LIN {X 0,Y 448.78,Z 726.193,A -85,B 0,C 180,E1 -8884.616,E2 -8884.616} C_VEL
LIN {X 0,Y 448.11,Z 736.801,A -85,B 0,C 180,E1 -8885.667,E2 -8885.667} C_VEL
LIN {X 0,Y 447.551,Z 746.669,A -85,B 0,C 180,E1 -8886.885,E2 -8886.885} C_VEL
LIN {X 0,Y 447.034,Z 755.083,A -85,B 0,C 180,E1 -8888.183,E2 -8888.183} C_VEL
LIN {X 0,Y 446.974,Z 755.977,A -85,B 0,C 180,E1 -8888.339,E2 -8888.339} C_VEL
LIN {X 0,Y 446.099,Z 759.432,A -85,B 0,C 180,E1 -8888.947,E2 -8888.947} C_VEL
LIN {X 0,Y 442.936,Z 764.696,A -85,B 0,C 180,E1 -8889.952,E2 -8889.952} C_VEL
LIN {X 0,Y 439.821,Z 769.35,A -85,B 0,C 180,E1 -8891.018,E2 -8891.018} C_VEL
LIN {X 0,Y 439.028,Z 771.716,A -85,B 0,C 180,E1 -8891.713,E2 -8891.713} C_VEL
LIN {X 0,Y 438.819,Z 775.806,A -85,B 0,C 180,E1 -8893.245,E2 -8893.245} C_VEL
LIN {X 0,Y 438.678,Z 777.727,A -85,B 0,C 180,E1 -8894.196,E2 -8894.196} C_VEL
LIN {X 0,Y 438.549,Z 779.208,A -85,B 0,C 180,E1 -8895.143,E2 -8895.143} C_VEL
LIN {X 0,Y 438.47,Z 780.829,A -85,B 0,C 180,E1 -8897.033,E2 -8897.033} C_VEL
LIN {X 0,Y 438.51,Z 781.044,A -85,B 0,C 180,E1 -8897.975,E2 -8897.975} C_VEL
LIN {X 0,Y 438.515,Z 780.818,A -85,B 0,C 180,E1 -8898.912,E2 -8898.912} C_VEL
LIN {X 0,Y 438.516,Z 779.204,A -85,B 0,C 180,E1 -8900.778,E2 -8900.778} C_VEL
LIN {X 0,Y 438.62,Z 777.768,A -85,B 0,C 180,E1 -8901.709,E2 -8901.709} C_VEL
LIN {X 0,Y 438.838,Z 774.591,A -85,B 0,C 180,E1 -8903.185,E2 -8903.185} C_VEL
LIN {X 0,Y 439.068,Z 769.268,A -85,B 0,C 180,E1 -8904.949,E2 -8904.949} C_VEL
LIN {X 0,Y 439.407,Z 762.676,A -85,B 0,C 180,E1 -8906.562,E2 -8906.562} C_VEL
LIN {X 0,Y 439.846,Z 755.516,A -85,B 0,C 180,E1 -8907.94,E2 -8907.94} C_VEL
LIN {X 0,Y 440.286,Z 748.225,A -85,B 0,C 180,E1 -8909.085,E2 -8909.085} C_VEL
LIN {X 0,Y 440.868,Z 739.403,A -85,B 0,C 180,E1 -8910.228,E2 -8910.228} C_VEL
LIN {X 0,Y 441.415,Z 728.463,A -85,B 0,C 180,E1 -8911.368,E2 -8911.368} C_VEL
LIN {X 0,Y 442.038,Z 717.473,A -85,B 0,C 180,E1 -8912.278,E2 -8912.278} C_VEL
LIN {X 0,Y 442.582,Z 705,A -85,B 0,C 180,E1 -8913.072,E2 -8913.072} C_VEL
LIN {X 0,Y 442.948,Z 692.395,A -85,B 0,C 180,E1 -8913.667,E2 -8913.667} C_VEL
LIN {X 0,Y 443.227,Z 680.1,A -85,B 0,C 180,E1 -8914.063,E2 -8914.063} C_VEL
LIN {X 0,Y 443.477,Z 656.155,A -85,B 0,C 180,E1 -8914.488,E2 -8914.488} C_VEL
LIN {X 0,Y 444.044,Z 588.908,A -85,B 0,C 180,E1 -8915.579,E2 -8915.579} C_VEL
LIN {X 0,Y 439.593,Z 575.73,A -85,B 0,C 180,E1 -8915.994,E2 -8915.994} C_VEL
LIN {X 0,Y 439.534,Z 575.738,A -85,B 0,C 180,E1 -8918.274,E2 -8918.274} C_VEL
LIN {X 0,Y 439.51,Z 575.741,A -85,B 0,C 180,E1 -8921.998,E2 -8921.998} C_VEL
LIN {X 0,Y 439.464,Z 575.743,A -85,B 0,C 180,E1 -8925.775,E2 -8925.775} C_VEL
LIN {X 0,Y 439.443,Z 575.743,A -85,B 0,C 180,E1 -8929.337,E2 -8929.337} C_VEL
LIN {X 0,Y 439.365,Z 575.754,A -85,B 0,C 180,E1 -8932.575,E2 -8932.575} C_VEL
LIN {X 0,Y 439.397,Z 575.751,A -85,B 0,C 180,E1 -8935.585,E2 -8935.585} C_VEL
LIN {X 0,Y 439.469,Z 575.744,A -85,B 0,C 180,E1 -8938.02,E2 -8938.02} C_VEL
LIN {X 0,Y 444.266,Z 589.404,A -85,B 0,C 180,E1 -8938.464,E2 -8938.464} C_VEL
LIN {X 0,Y 443.152,Z 678.564,A -85,B 0,C 180,E1 -8939.987,E2 -8939.987} C_VEL
LIN {X 0,Y 442.929,Z 692.439,A -85,B 0,C 180,E1 -8940.431,E2 -8940.431} C_VEL
LIN {X 0,Y 442.524,Z 705.387,A -85,B 0,C 180,E1 -8941.049,E2 -8941.049} C_VEL
LIN {X 0,Y 442.045,Z 716.757,A -85,B 0,C 180,E1 -8941.778,E2 -8941.778} C_VEL
LIN {X 0,Y 441.489,Z 728.769,A -85,B 0,C 180,E1 -8942.767,E2 -8942.767} C_VEL
LIN {X 0,Y 440.928,Z 738.453,A -85,B 0,C 180,E1 -8943.77,E2 -8943.77} C_VEL
LIN {X 0,Y 440.317,Z 748.569,A -85,B 0,C 180,E1 -8945.071,E2 -8945.071} C_VEL
LIN {X 0,Y 439.875,Z 755.956,A -85,B 0,C 180,E1 -8946.238,E2 -8946.238} C_VEL
LIN {X 0,Y 439.396,Z 763.311,A -85,B 0,C 180,E1 -8947.662,E2 -8947.662} C_VEL
LIN {X 0,Y 439.083,Z 769.474,A -85,B 0,C 180,E1 -8949.192,E2 -8949.192} C_VEL
LIN {X 0,Y 438.838,Z 773.436,A -85,B 0,C 180,E1 -8950.436,E2 -8950.436} C_VEL
LIN {X 0,Y 438.69,Z 776.55,A -85,B 0,C 180,E1 -8951.69,E2 -8951.69} C_VEL
LIN {X 0,Y 438.577,Z 778.129,A -85,B 0,C 180,E1 -8952.512,E2 -8952.512} C_VEL
LIN {X 0,Y 438.477,Z 779.994,A -85,B 0,C 180,E1 -8953.84,E2 -8953.84} C_VEL
LIN {X 0,Y 438.416,Z 780.98,A -85,B 0,C 180,E1 -8955.143,E2 -8955.143} C_VEL
LIN {X 0,Y 438.403,Z 781.18,A -85,B 0,C 180,E1 -8956.423,E2 -8956.423} C_VEL
LIN {X 0,Y 438.468,Z 780.644,A -85,B 0,C 180,E1 -8957.685,E2 -8957.685} C_VEL
LIN {X 0,Y 438.56,Z 779.387,A -85,B 0,C 180,E1 -8958.926,E2 -8958.926} C_VEL
LIN {X 0,Y 438.764,Z 775.998,A -85,B 0,C 180,E1 -8960.807,E2 -8960.807} C_VEL
LIN {X 0,Y 439.01,Z 772.573,A -85,B 0,C 180,E1 -8962.11,E2 -8962.11} C_VEL
LIN {X 0,Y 439.311,Z 767.045,A -85,B 0,C 180,E1 -8963.707,E2 -8963.707} C_VEL
LIN {X 0,Y 439.69,Z 760.584,A -85,B 0,C 180,E1 -8965.15,E2 -8965.15} C_VEL
LIN {X 0,Y 440.113,Z 753.59,A -85,B 0,C 180,E1 -8966.403,E2 -8966.403} C_VEL
LIN {X 0,Y 440.746,Z 744.764,A -85,B 0,C 180,E1 -8967.683,E2 -8967.683} C_VEL
LIN {X 0,Y 441.288,Z 735.189,A -85,B 0,C 180,E1 -8968.814,E2 -8968.814} C_VEL
LIN {X 0,Y 441.891,Z 724.799,A -85,B 0,C 180,E1 -8969.803,E2 -8969.803} C_VEL
LIN {X 0,Y 442.376,Z 714.046,A -85,B 0,C 180,E1 -8970.619,E2 -8970.619} C_VEL
LIN {X 0,Y 442.917,Z 701.443,A -85,B 0,C 180,E1 -8971.355,E2 -8971.355} C_VEL
LIN {X 0,Y 443.186,Z 688.797,A -85,B 0,C 180,E1 -8971.893,E2 -8971.893} C_VEL
LIN {X 0,Y 443.426,Z 676.012,A -85,B 0,C 180,E1 -8972.239,E2 -8972.239} C_VEL
LIN {X 0,Y 444.343,Z 588.817,A -85,B 0,C 180,E1 -8973.74,E2 -8973.74} C_VEL
LIN {X 0,Y 439.477,Z 575.744,A -85,B 0,C 180,E1 -8974.203,E2 -8974.203} C_VEL
LIN {X 0,Y 439.357,Z 575.757,A -85,B 0,C 180,E1 -8977.424,E2 -8977.424} C_VEL
LIN {X 0,Y 439.433,Z 575.75,A -85,B 0,C 180,E1 -8980.662,E2 -8980.662} C_VEL
LIN {X 0,Y 439.453,Z 575.747,A -85,B 0,C 180,E1 -8984.224,E2 -8984.224} C_VEL
LIN {X 0,Y 439.503,Z 575.739,A -85,B 0,C 180,E1 -8988.002,E2 -8988.002} C_VEL
LIN {X 0,Y 439.539,Z 575.732,A -85,B 0,C 180,E1 -8991.726,E2 -8991.726} C_VEL
LIN {X 0,Y 439.618,Z 575.726,A -85,B 0,C 180,E1 -8994.496,E2 -8994.496} C_VEL
LIN {X 0,Y 439.626,Z 575.721,A -85,B 0,C 180,E1 -8998.168,E2 -8998.168} C_VEL
LIN {X 0,Y 439.755,Z 575.706,A -85,B 0,C 180,E1 -9000,E2 -9000} C_VEL
LIN {X 0,Y 439.648,Z 575.719,A -85,B 0,C 180,E1 -9002.749,E2 -9002.749} C_VEL
LIN {X 0,Y 439.613,Z 575.724,A -85,B 0,C 180,E1 -9006.425,E2 -9006.425} C_VEL
LIN {X 0,Y 439.492,Z 575.734,A -85,B 0,C 180,E1 -9009.202,E2 -9009.202} C_VEL
LIN {X 0,Y 439.495,Z 575.734,A -85,B 0,C 180,E1 -9012.727,E2 -9012.727} C_VEL
LIN {X 0,Y 439.438,Z 575.744,A -85,B 0,C 180,E1 -9016.349,E2 -9016.349} C_VEL
LIN {X 0,Y 439.395,Z 575.745,A -85,B 0,C 180,E1 -9019.627,E2 -9019.627} C_VEL
LIN {X 0,Y 439.359,Z 575.757,A -85,B 0,C 180,E1 -9022.576,E2 -9022.576} C_VEL
LIN {X 0,Y 439.398,Z 575.748,A -85,B 0,C 180,E1 -9025.585,E2 -9025.585} C_VEL
LIN {X 0,Y 439.418,Z 575.752,A -85,B 0,C 180,E1 -9028.674,E2 -9028.674} C_VEL
LIN {X 0,Y 439.368,Z 575.753,A -85,B 0,C 180,E1 -9031.861,E2 -9031.861} C_VEL
LIN {X 0,Y 439.395,Z 575.75,A -85,B 0,C 180,E1 -9035.157,E2 -9035.157} C_VEL
LIN {X 0,Y 439.394,Z 575.753,A -85,B 0,C 180,E1 -9038.594,E2 -9038.594} C_VEL
LIN {X 0,Y 439.4,Z 575.747,A -85,B 0,C 180,E1 -9041.26,E2 -9041.26} C_VEL
LIN {X 0,Y 439.404,Z 575.754,A -85,B 0,C 180,E1 -9044.729,E2 -9044.729} C_VEL
LIN {X 0,Y 439.393,Z 575.751,A -85,B 0,C 180,E1 -9047.797,E2 -9047.797} C_VEL
LIN {X 0,Y 439.448,Z 575.747,A -85,B 0,C 180,E1 -9050.231,E2 -9050.231} C_VEL
LIN {X 0,Y 439.374,Z 575.753,A -85,B 0,C 180,E1 -9053.714,E2 -9053.714} C_VEL
LIN {X 0,Y 439.371,Z 575.755,A -85,B 0,C 180,E1 -9057.055,E2 -9057.055} C_VEL
LIN {X 0,Y 439.443,Z 575.82,A -85,B 0,C 180,E1 -9060.707,E2 -9060.707} C_VEL
LIN {X 0,Y 442.42,Z 589.659,A -85,B 0,C 180,E1 -9063.274,E2 -9063.274} C_VEL
LIN {X 0,Y 442.893,Z 594.558,A -85,B 0,C 180,E1 -9064.128,E2 -9064.128} C_VEL
LIN {X 0,Y 441.873,Z 612.173,A -85,B 0,C 180,E1 -9067.021,E2 -9067.021} C_VEL
LIN {X 0,Y 440.837,Z 633.371,A -85,B 0,C 180,E1 -9070.441,E2 -9070.441} C_VEL
LIN {X 0,Y 440.413,Z 641.915,A -85,B 0,C 180,E1 -9071.806,E2 -9071.806} C_VEL
LIN {X 0,Y 443.891,Z 669.193,A -85,B 0,C 180,E1 -9072.436,E2 -9072.436} C_VEL
LIN {X 0,Y 442.998,Z 751.905,A -85,B 0,C 180,E1 -9073.852,E2 -9073.852} C_VEL
LIN {X 0,Y 442.553,Z 765.081,A -85,B 0,C 180,E1 -9074.249,E2 -9074.249} C_VEL
LIN {X 0,Y 442.027,Z 776.143,A -85,B 0,C 180,E1 -9074.732,E2 -9074.732} C_VEL
LIN {X 0,Y 441.373,Z 788.842,A -85,B 0,C 180,E1 -9075.476,E2 -9075.476} C_VEL
LIN {X 0,Y 440.764,Z 800.147,A -85,B 0,C 180,E1 -9076.344,E2 -9076.344} C_VEL
LIN {X 0,Y 440.178,Z 811.45,A -85,B 0,C 180,E1 -9077.436,E2 -9077.436} C_VEL
LIN {X 0,Y 439.622,Z 820.217,A -85,B 0,C 180,E1 -9078.473,E2 -9078.473} C_VEL
LIN {X 0,Y 439.176,Z 828.317,A -85,B 0,C 180,E1 -9079.629,E2 -9079.629} C_VEL
LIN {X 0,Y 438.816,Z 836.256,A -85,B 0,C 180,E1 -9081.016,E2 -9081.016} C_VEL
LIN {X 0,Y 438.608,Z 843.573,A -85,B 0,C 180,E1 -9082.635,E2 -9082.635} C_VEL
LIN {X 0,Y 438.479,Z 847.975,A -85,B 0,C 180,E1 -9083.869,E2 -9083.869} C_VEL
LIN {X 0,Y 438.401,Z 852.206,A -85,B 0,C 180,E1 -9085.403,E2 -9085.403} C_VEL
LIN {X 0,Y 438.479,Z 854.154,A -85,B 0,C 180,E1 -9086.324,E2 -9086.324} C_VEL
LIN {X 0,Y 438.509,Z 855.616,A -85,B 0,C 180,E1 -9087.244,E2 -9087.244} C_VEL
LIN {X 0,Y 438.466,Z 856.659,A -85,B 0,C 180,E1 -9088.163,E2 -9088.163} C_VEL
LIN {X 0,Y 438.381,Z 857.299,A -85,B 0,C 180,E1 -9089.081,E2 -9089.081} C_VEL
LIN {X 0,Y 438.361,Z 857.538,A -85,B 0,C 180,E1 -9090,E2 -9090} C_VEL
LIN {X 0,Y 438.466,Z 856.734,A -85,B 0,C 180,E1 -9091.837,E2 -9091.837} C_VEL
LIN {X 0,Y 438.508,Z 855.731,A -85,B 0,C 180,E1 -9092.756,E2 -9092.756} C_VEL
LIN {X 0,Y 438.476,Z 854.299,A -85,B 0,C 180,E1 -9093.676,E2 -9093.676} C_VEL
LIN {X 0,Y 438.453,Z 851.302,A -85,B 0,C 180,E1 -9095.058,E2 -9095.058} C_VEL
LIN {X 0,Y 438.506,Z 847.237,A -85,B 0,C 180,E1 -9096.441,E2 -9096.441} C_VEL
LIN {X 0,Y 438.671,Z 840.963,A -85,B 0,C 180,E1 -9098.058,E2 -9098.058} C_VEL
LIN {X 0,Y 438.909,Z 834.122,A -85,B 0,C 180,E1 -9099.446,E2 -9099.446} C_VEL
LIN {X 0,Y 439.357,Z 825.638,A -85,B 0,C 180,E1 -9100.833,E2 -9100.833} C_VEL
LIN {X 0,Y 439.809,Z 816.892,A -85,B 0,C 180,E1 -9101.989,E2 -9101.989} C_VEL
LIN {X 0,Y 440.399,Z 806.912,A -85,B 0,C 180,E1 -9103.068,E2 -9103.068} C_VEL
LIN {X 0,Y 441.032,Z 795.466,A -85,B 0,C 180,E1 -9104.064,E2 -9104.064} C_VEL
LIN {X 0,Y 441.689,Z 783.61,A -85,B 0,C 180,E1 -9104.867,E2 -9104.867} C_VEL
LIN {X 0,Y 442.214,Z 771.308,A -85,B 0,C 180,E1 -9105.497,E2 -9105.497} C_VEL
LIN {X 0,Y 442.8,Z 757.864,A -85,B 0,C 180,E1 -9105.978,E2 -9105.978} C_VEL
LIN {X 0,Y 443.127,Z 742.721,A -85,B 0,C 180,E1 -9106.291,E2 -9106.291} C_VEL
LIN {X 0,Y 443.758,Z 666.118,A -85,B 0,C 180,E1 -9107.584,E2 -9107.584} C_VEL
LIN {X 0,Y 440.913,Z 642.526,A -85,B 0,C 180,E1 -9108.115,E2 -9108.115} C_VEL
LIN {X 0,Y 441.932,Z 622.104,A -85,B 0,C 180,E1 -9110.966,E2 -9110.966} C_VEL
LIN {X 0,Y 443.256,Z 598.165,A -85,B 0,C 180,E1 -9114.345,E2 -9114.345} C_VEL
LIN {X 0,Y 443.448,Z 594.812,A -85,B 0,C 180,E1 -9114.822,E2 -9114.822} C_VEL
LIN {X 0,Y 441.817,Z 585.976,A -85,B 0,C 180,E1 -9116.194,E2 -9116.194} C_VEL
LIN {X 0,Y 439.473,Z 575.746,A -85,B 0,C 180,E1 -9117.866,E2 -9117.866} C_VEL
LIN {X 0,Y 439.36,Z 575.755,A -85,B 0,C 180,E1 -9120.788,E2 -9120.788} C_VEL
LIN {X 0,Y 439.386,Z 575.756,A -85,B 0,C 180,E1 -9124.043,E2 -9124.043} C_VEL
LIN {X 0,Y 439.361,Z 575.755,A -85,B 0,C 180,E1 -9127.433,E2 -9127.433} C_VEL
LIN {X 0,Y 439.423,Z 575.749,A -85,B 0,C 180,E1 -9129.852,E2 -9129.852} C_VEL
LIN {X 0,Y 439.378,Z 575.752,A -85,B 0,C 180,E1 -9132.626,E2 -9132.626} C_VEL
LIN {X 0,Y 439.399,Z 575.748,A -85,B 0,C 180,E1 -9136.033,E2 -9136.033} C_VEL
LIN {X 0,Y 439.395,Z 575.747,A -85,B 0,C 180,E1 -9139.021,E2 -9139.021} C_VEL
LIN {X 0,Y 439.387,Z 575.747,A -85,B 0,C 180,E1 -9141.604,E2 -9141.604} C_VEL
LIN {X 0,Y 439.394,Z 575.741,A -85,B 0,C 180,E1 -9144.843,E2 -9144.843} C_VEL
LIN {X 0,Y 439.381,Z 575.755,A -85,B 0,C 180,E1 -9148.14,E2 -9148.14} C_VEL
LIN {X 0,Y 439.418,Z 575.736,A -85,B 0,C 180,E1 -9151.326,E2 -9151.326} C_VEL
LIN {X 0,Y 439.398,Z 575.754,A -85,B 0,C 180,E1 -9154.415,E2 -9154.415} C_VEL
LIN {X 0,Y 439.356,Z 575.742,A -85,B 0,C 180,E1 -9157.424,E2 -9157.424} C_VEL
LIN {X 0,Y 439.433,Z 575.748,A -85,B 0,C 180,E1 -9160.662,E2 -9160.662} C_VEL
LIN {X 0,Y 439.453,Z 575.734,A -85,B 0,C 180,E1 -9164.224,E2 -9164.224} C_VEL
LIN {X 0,Y 439.475,Z 575.74,A -85,B 0,C 180,E1 -9168.001,E2 -9168.001} C_VEL
LIN {X 0,Y 439.538,Z 575.72,A -85,B 0,C 180,E1 -9171.726,E2 -9171.726} C_VEL
LIN {X 0,Y 439.619,Z 575.725,A -85,B 0,C 180,E1 -9174.496,E2 -9174.496} C_VEL
LIN {X 0,Y 439.627,Z 575.712,A -85,B 0,C 180,E1 -9178.168,E2 -9178.168} C_VEL
LIN {X 0,Y 439.755,Z 575.698,A -85,B 0,C 180,E1 -9180,E2 -9180} C_VEL
LIN {X 0,Y 439.648,Z 575.722,A -85,B 0,C 180,E1 -9182.749,E2 -9182.749} C_VEL
LIN {X 0,Y 439.611,Z 575.712,A -85,B 0,C 180,E1 -9186.425,E2 -9186.425} C_VEL
LIN {X 0,Y 439.491,Z 575.739,A -85,B 0,C 180,E1 -9189.202,E2 -9189.202} C_VEL
LIN {X 0,Y 439.457,Z 575.736,A -85,B 0,C 180,E1 -9192.938,E2 -9192.938} C_VEL
LIN {X 0,Y 439.438,Z 575.744,A -85,B 0,C 180,E1 -9196.349,E2 -9196.349} C_VEL
LIN {X 0,Y 439.394,Z 575.745,A -85,B 0,C 180,E1 -9199.627,E2 -9199.627} C_VEL
LIN {X 0,Y 439.356,Z 575.756,A -85,B 0,C 180,E1 -9202.576,E2 -9202.576} C_VEL
LIN {X 0,Y 439.398,Z 575.748,A -85,B 0,C 180,E1 -9205.585,E2 -9205.585} C_VEL
LIN {X 0,Y 439.418,Z 575.748,A -85,B 0,C 180,E1 -9208.674,E2 -9208.674} C_VEL
LIN {X 0,Y 439.378,Z 575.751,A -85,B 0,C 180,E1 -9212.034,E2 -9212.034} C_VEL
LIN {X 0,Y 439.39,Z 575.753,A -85,B 0,C 180,E1 -9215.341,E2 -9215.341} C_VEL
LIN {X 0,Y 439.387,Z 575.751,A -85,B 0,C 180,E1 -9218.595,E2 -9218.595} C_VEL
LIN {X 0,Y 439.393,Z 575.738,A -85,B 0,C 180,E1 -9221.259,E2 -9221.259} C_VEL
LIN {X 0,Y 439.401,Z 575.749,A -85,B 0,C 180,E1 -9224.73,E2 -9224.73} C_VEL
LIN {X 0,Y 439.392,Z 575.742,A -85,B 0,C 180,E1 -9227.796,E2 -9227.796} C_VEL
LIN {X 0,Y 439.423,Z 575.746,A -85,B 0,C 180,E1 -9230.228,E2 -9230.228} C_VEL
LIN {X 0,Y 439.375,Z 575.756,A -85,B 0,C 180,E1 -9233.714,E2 -9233.714} C_VEL
LIN {X 0,Y 439.371,Z 575.756,A -85,B 0,C 180,E1 -9237.055,E2 -9237.055} C_VEL
LIN {X 0,Y 439.39,Z 575.754,A -85,B 0,C 180,E1 -9239.824,E2 -9239.824} C_VEL
LIN {X 0,Y 441.332,Z 580.971,A -85,B 0,C 180,E1 -9240.019,E2 -9240.019} C_VEL
LIN {X 0,Y 444.652,Z 589.408,A -85,B 0,C 180,E1 -9240.32,E2 -9240.32} C_VEL
LIN {X 0,Y 443.622,Z 677.951,A -85,B 0,C 180,E1 -9241.785,E2 -9241.785} C_VEL
LIN {X 0,Y 443.413,Z 690.45,A -85,B 0,C 180,E1 -9242.156,E2 -9242.156} C_VEL
LIN {X 0,Y 443.099,Z 702.807,A -85,B 0,C 180,E1 -9242.706,E2 -9242.706} C_VEL
LIN {X 0,Y 442.623,Z 713.699,A -85,B 0,C 180,E1 -9243.357,E2 -9243.357} C_VEL
LIN {X 0,Y 442.044,Z 724.739,A -85,B 0,C 180,E1 -9244.201,E2 -9244.201} C_VEL
LIN {X 0,Y 441.44,Z 734.788,A -85,B 0,C 180,E1 -9245.159,E2 -9245.159} C_VEL
LIN {X 0,Y 440.852,Z 744.173,A -85,B 0,C 180,E1 -9246.264,E2 -9246.264} C_VEL
LIN {X 0,Y 440.29,Z 752.531,A -85,B 0,C 180,E1 -9247.475,E2 -9247.475} C_VEL
LIN {X 0,Y 439.771,Z 760.635,A -85,B 0,C 180,E1 -9248.927,E2 -9248.927} C_VEL
LIN {X 0,Y 439.339,Z 767.04,A -85,B 0,C 180,E1 -9250.371,E2 -9250.371} C_VEL
LIN {X 0,Y 439.028,Z 771.716,A -85,B 0,C 180,E1 -9251.713,E2 -9251.713} C_VEL
LIN {X 0,Y 438.246,Z 773.899,A -85,B 0,C 180,E1 -9252.423,E2 -9252.423} C_VEL
LIN {X 0,Y 435.194,Z 776.991,A -85,B 0,C 180,E1 -9253.594,E2 -9253.594} C_VEL
LIN {X 0,Y 432.653,Z 778.955,A -85,B 0,C 180,E1 -9254.558,E2 -9254.558} C_VEL
LIN {X 0,Y 431.552,Z 780.087,A -85,B 0,C 180,E1 -9255.316,E2 -9255.316} C_VEL
LIN {X 0,Y 431.456,Z 780.354,A -85,B 0,C 180,E1 -9255.575,E2 -9255.575} C_VEL
LIN {X 0,Y 431.395,Z 781.35,A -85,B 0,C 180,E1 -9256.816,E2 -9256.816} C_VEL
LIN {X 0,Y 431.433,Z 781.628,A -85,B 0,C 180,E1 -9257.795,E2 -9257.795} C_VEL
LIN {X 0,Y 431.445,Z 781.506,A -85,B 0,C 180,E1 -9258.728,E2 -9258.728} C_VEL
LIN {X 0,Y 431.437,Z 780.007,A -85,B 0,C 180,E1 -9260.625,E2 -9260.625} C_VEL
LIN {X 0,Y 431.529,Z 778.669,A -85,B 0,C 180,E1 -9261.572,E2 -9261.572} C_VEL
LIN {X 0,Y 431.778,Z 775.393,A -85,B 0,C 180,E1 -9263.165,E2 -9263.165} C_VEL
LIN {X 0,Y 432.001,Z 770.432,A -85,B 0,C 180,E1 -9264.867,E2 -9264.867} C_VEL
LIN {X 0,Y 432.273,Z 765.064,A -85,B 0,C 180,E1 -9266.271,E2 -9266.271} C_VEL
LIN {X 0,Y 432.739,Z 758.341,A -85,B 0,C 180,E1 -9267.673,E2 -9267.673} C_VEL
LIN {X 0,Y 433.251,Z 749.932,A -85,B 0,C 180,E1 -9269.071,E2 -9269.071} C_VEL
LIN {X 0,Y 433.838,Z 741.33,A -85,B 0,C 180,E1 -9270.232,E2 -9270.232} C_VEL
LIN {X 0,Y 434.416,Z 730.777,A -85,B 0,C 180,E1 -9271.391,E2 -9271.391} C_VEL
LIN {X 0,Y 435.012,Z 720.168,A -85,B 0,C 180,E1 -9272.315,E2 -9272.315} C_VEL
LIN {X 0,Y 435.616,Z 708.398,A -85,B 0,C 180,E1 -9273.121,E2 -9273.121} C_VEL
LIN {X 0,Y 436.035,Z 696.124,A -85,B 0,C 180,E1 -9273.754,E2 -9273.754} C_VEL
LIN {X 0,Y 436.328,Z 683.342,A -85,B 0,C 180,E1 -9274.214,E2 -9274.214} C_VEL
LIN {X 0,Y 436.484,Z 670.113,A -85,B 0,C 180,E1 -9274.502,E2 -9274.502} C_VEL
LIN {X 0,Y 437.208,Z 590.4,A -85,B 0,C 180,E1 -9275.814,E2 -9275.814} C_VEL
LIN {X 0,Y 432.558,Z 576.606,A -85,B 0,C 180,E1 -9276.238,E2 -9276.238} C_VEL
LIN {X 0,Y 432.443,Z 576.617,A -85,B 0,C 180,E1 -9279.353,E2 -9279.353} C_VEL
LIN {X 0,Y 432.447,Z 576.614,A -85,B 0,C 180,E1 -9282.811,E2 -9282.811} C_VEL
LIN {X 0,Y 432.414,Z 576.621,A -85,B 0,C 180,E1 -9286.479,E2 -9286.479} C_VEL
LIN {X 0,Y 432.34,Z 576.634,A -85,B 0,C 180,E1 -9289.96,E2 -9289.96} C_VEL
LIN {X 0,Y 432.318,Z 576.63,A -85,B 0,C 180,E1 -9292.964,E2 -9292.964} C_VEL
LIN {X 0,Y 432.358,Z 576.631,A -85,B 0,C 180,E1 -9296.032,E2 -9296.032} C_VEL
LIN {X 0,Y 432.42,Z 576.624,A -85,B 0,C 180,E1 -9297.725,E2 -9297.725} C_VEL
LIN {X 0,Y 437.447,Z 590.525,A -85,B 0,C 180,E1 -9298.204,E2 -9298.204} C_VEL
LIN {X 0,Y 436.321,Z 678.909,A -85,B 0,C 180,E1 -9299.739,E2 -9299.739} C_VEL
LIN {X 0,Y 436.103,Z 692.378,A -85,B 0,C 180,E1 -9300.171,E2 -9300.171} C_VEL
LIN {X 0,Y 435.775,Z 704.32,A -85,B 0,C 180,E1 -9300.732,E2 -9300.732} C_VEL
LIN {X 0,Y 435.217,Z 716.576,A -85,B 0,C 180,E1 -9301.509,E2 -9301.509} C_VEL
LIN {X 0,Y 434.643,Z 728.421,A -85,B 0,C 180,E1 -9302.484,E2 -9302.484} C_VEL
LIN {X 0,Y 434.015,Z 738.678,A -85,B 0,C 180,E1 -9303.544,E2 -9303.544} C_VEL
LIN {X 0,Y 433.375,Z 748.854,A -85,B 0,C 180,E1 -9304.864,E2 -9304.864} C_VEL
LIN {X 0,Y 432.904,Z 756.297,A -85,B 0,C 180,E1 -9306.05,E2 -9306.05} C_VEL
LIN {X 0,Y 432.488,Z 762.422,A -85,B 0,C 180,E1 -9307.226,E2 -9307.226} C_VEL
LIN {X 0,Y 432.159,Z 768.599,A -85,B 0,C 180,E1 -9308.684,E2 -9308.684} C_VEL
LIN {X 0,Y 431.831,Z 773.318,A -85,B 0,C 180,E1 -9310.1,E2 -9310.1} C_VEL
LIN {X 0,Y 431.655,Z 776.866,A -85,B 0,C 180,E1 -9311.5,E2 -9311.5} C_VEL
LIN {X 0,Y 431.455,Z 779.814,A -85,B 0,C 180,E1 -9313.167,E2 -9313.167} C_VEL
LIN {X 0,Y 431.379,Z 781.197,A -85,B 0,C 180,E1 -9314.47,E2 -9314.47} C_VEL
LIN {X 0,Y 431.337,Z 781.794,A -85,B 0,C 180,E1 -9315.799,E2 -9315.799} C_VEL
LIN {X 0,Y 431.365,Z 781.591,A -85,B 0,C 180,E1 -9317.15,E2 -9317.15} C_VEL
LIN {X 0,Y 431.47,Z 780.535,A -85,B 0,C 180,E1 -9318.526,E2 -9318.526} C_VEL
LIN {X 0,Y 431.587,Z 778.541,A -85,B 0,C 180,E1 -9319.937,E2 -9319.937} C_VEL
LIN {X 0,Y 431.836,Z 775.511,A -85,B 0,C 180,E1 -9321.367,E2 -9321.367} C_VEL
LIN {X 0,Y 432.12,Z 770.708,A -85,B 0,C 180,E1 -9323.003,E2 -9323.003} C_VEL
LIN {X 0,Y 432.499,Z 764.489,A -85,B 0,C 180,E1 -9324.606,E2 -9324.606} C_VEL
LIN {X 0,Y 432.933,Z 758.219,A -85,B 0,C 180,E1 -9325.882,E2 -9325.882} C_VEL
LIN {X 0,Y 433.52,Z 749.749,A -85,B 0,C 180,E1 -9327.271,E2 -9327.271} C_VEL
LIN {X 0,Y 434.118,Z 740.269,A -85,B 0,C 180,E1 -9328.527,E2 -9328.527} C_VEL
LIN {X 0,Y 434.707,Z 731.039,A -85,B 0,C 180,E1 -9329.519,E2 -9329.519} C_VEL
LIN {X 0,Y 435.358,Z 719.709,A -85,B 0,C 180,E1 -9330.496,E2 -9330.496} C_VEL
LIN {X 0,Y 435.829,Z 708.333,A -85,B 0,C 180,E1 -9331.266,E2 -9331.266} C_VEL
LIN {X 0,Y 436.292,Z 696.129,A -85,B 0,C 180,E1 -9331.889,E2 -9331.889} C_VEL
LIN {X 0,Y 436.551,Z 683.948,A -85,B 0,C 180,E1 -9332.328,E2 -9332.328} C_VEL
LIN {X 0,Y 436.743,Z 667.683,A -85,B 0,C 180,E1 -9332.67,E2 -9332.67} C_VEL
LIN {X 0,Y 437.646,Z 590.35,A -85,B 0,C 180,E1 -9334.017,E2 -9334.017} C_VEL
LIN {X 0,Y 432.577,Z 577.468,A -85,B 0,C 180,E1 -9334.498,E2 -9334.498} C_VEL
LIN {X 0,Y 432.396,Z 576.627,A -85,B 0,C 180,E1 -9334.551,E2 -9334.551} C_VEL
LIN {X 0,Y 432.349,Z 576.63,A -85,B 0,C 180,E1 -9338.045,E2 -9338.045} C_VEL
LIN {X 0,Y 432.378,Z 576.627,A -85,B 0,C 180,E1 -9341.029,E2 -9341.029} C_VEL
LIN {X 0,Y 432.421,Z 576.62,A -85,B 0,C 180,E1 -9343.961,E2 -9343.961} C_VEL
LIN {X 0,Y 432.475,Z 576.613,A -85,B 0,C 180,E1 -9347.804,E2 -9347.804} C_VEL
LIN {X 0,Y 432.483,Z 576.611,A -85,B 0,C 180,E1 -9351.59,E2 -9351.59} C_VEL
LIN {X 0,Y 432.594,Z 576.601,A -85,B 0,C 180,E1 -9354.406,E2 -9354.406} C_VEL
LIN {X 0,Y 432.596,Z 576.596,A -85,B 0,C 180,E1 -9358.138,E2 -9358.138} C_VEL
LIN {X 0,Y 432.725,Z 576.582,A -85,B 0,C 180,E1 -9360,E2 -9360} C_VEL
LIN {X 0,Y 432.597,Z 576.596,A -85,B 0,C 180,E1 -9362.794,E2 -9362.794} C_VEL
LIN {X 0,Y 432.567,Z 576.6,A -85,B 0,C 180,E1 -9366.53,E2 -9366.53} C_VEL
LIN {X 0,Y 432.436,Z 576.612,A -85,B 0,C 180,E1 -9369.353,E2 -9369.353} C_VEL
LIN {X 0,Y 432.436,Z 576.612,A -85,B 0,C 180,E1 -9372.812,E2 -9372.812} C_VEL
LIN {X 0,Y 432.403,Z 576.619,A -85,B 0,C 180,E1 -9376.479,E2 -9376.479} C_VEL
LIN {X 0,Y 432.333,Z 576.627,A -85,B 0,C 180,E1 -9379.961,E2 -9379.961} C_VEL
LIN {X 0,Y 432.313,Z 576.63,A -85,B 0,C 180,E1 -9382.965,E2 -9382.965} C_VEL
LIN {X 0,Y 432.357,Z 576.628,A -85,B 0,C 180,E1 -9386.033,E2 -9386.033} C_VEL
LIN {X 0,Y 432.345,Z 576.628,A -85,B 0,C 180,E1 -9389.187,E2 -9389.187} C_VEL
LIN {X 0,Y 432.319,Z 576.635,A -85,B 0,C 180,E1 -9392.294,E2 -9392.294} C_VEL
LIN {X 0,Y 432.335,Z 576.634,A -85,B 0,C 180,E1 -9394.678,E2 -9394.678} C_VEL
LIN {X 0,Y 432.348,Z 576.63,A -85,B 0,C 180,E1 -9398.149,E2 -9398.149} C_VEL
LIN {X 0,Y 432.368,Z 576.623,A -85,B 0,C 180,E1 -9401.609,E2 -9401.609} C_VEL
LIN {X 0,Y 432.374,Z 576.628,A -85,B 0,C 180,E1 -9404.342,E2 -9404.342} C_VEL
LIN {X 0,Y 432.363,Z 576.631,A -85,B 0,C 180,E1 -9408.394,E2 -9408.394} C_VEL
LIN {X 0,Y 432.349,Z 576.629,A -85,B 0,C 180,E1 -9411.852,E2 -9411.852} C_VEL
LIN {X 0,Y 432.338,Z 576.63,A -85,B 0,C 180,E1 -9415.324,E2 -9415.324} C_VEL
LIN {X 0,Y 432.32,Z 576.635,A -85,B 0,C 180,E1 -9418.655,E2 -9418.655} C_VEL
LIN {X 0,Y 432.392,Z 576.678,A -85,B 0,C 180,E1 -9420.416,E2 -9420.416} C_VEL
LIN {X 0,Y 435.48,Z 591.029,A -85,B 0,C 180,E1 -9423.136,E2 -9423.136} C_VEL
LIN {X 0,Y 436.001,Z 595.554,A -85,B 0,C 180,E1 -9423.945,E2 -9423.945} C_VEL
LIN {X 0,Y 434.857,Z 614.484,A -85,B 0,C 180,E1 -9427.105,E2 -9427.105} C_VEL
LIN {X 0,Y 433.821,Z 634.276,A -85,B 0,C 180,E1 -9430.358,E2 -9430.358} C_VEL
LIN {X 0,Y 433.449,Z 641.208,A -85,B 0,C 180,E1 -9431.483,E2 -9431.483} C_VEL
LIN {X 0,Y 437.132,Z 669.77,A -85,B 0,C 180,E1 -9432.163,E2 -9432.163} C_VEL
LIN {X 0,Y 436.179,Z 751.494,A -85,B 0,C 180,E1 -9433.592,E2 -9433.592} C_VEL
LIN {X 0,Y 435.697,Z 765.314,A -85,B 0,C 180,E1 -9434.025,E2 -9434.025} C_VEL
LIN {X 0,Y 435.105,Z 776.693,A -85,B 0,C 180,E1 -9434.543,E2 -9434.543} C_VEL
LIN {X 0,Y 434.493,Z 788.221,A -85,B 0,C 180,E1 -9435.241,E2 -9435.241} C_VEL
LIN {X 0,Y 433.793,Z 800.016,A -85,B 0,C 180,E1 -9436.167,E2 -9436.167} C_VEL
LIN {X 0,Y 433.231,Z 810.814,A -85,B 0,C 180,E1 -9437.231,E2 -9437.231} C_VEL
LIN {X 0,Y 432.615,Z 819.581,A -85,B 0,C 180,E1 -9438.284,E2 -9438.284} C_VEL
LIN {X 0,Y 432.143,Z 827.685,A -85,B 0,C 180,E1 -9439.458,E2 -9439.458} C_VEL
LIN {X 0,Y 431.756,Z 835.625,A -85,B 0,C 180,E1 -9440.868,E2 -9440.868} C_VEL
LIN {X 0,Y 431.569,Z 841.068,A -85,B 0,C 180,E1 -9442.044,E2 -9442.044} C_VEL
LIN {X 0,Y 431.396,Z 846.829,A -85,B 0,C 180,E1 -9443.603,E2 -9443.603} C_VEL
LIN {X 0,Y 431.394,Z 850.479,A -85,B 0,C 180,E1 -9444.859,E2 -9444.859} C_VEL
LIN {X 0,Y 431.383,Z 853.536,A -85,B 0,C 180,E1 -9446.264,E2 -9446.264} C_VEL
LIN {X 0,Y 431.432,Z 854.999,A -85,B 0,C 180,E1 -9447.199,E2 -9447.199} C_VEL
LIN {X 0,Y 431.411,Z 856.044,A -85,B 0,C 180,E1 -9448.133,E2 -9448.133} C_VEL
LIN {X 0,Y 431.322,Z 856.685,A -85,B 0,C 180,E1 -9449.066,E2 -9449.066} C_VEL
LIN {X 0,Y 431.3,Z 856.921,A -85,B 0,C 180,E1 -9450,E2 -9450} C_VEL
LIN {X 0,Y 431.411,Z 856.114,A -85,B 0,C 180,E1 -9451.867,E2 -9451.867} C_VEL
LIN {X 0,Y 431.431,Z 855.106,A -85,B 0,C 180,E1 -9452.801,E2 -9452.801} C_VEL
LIN {X 0,Y 431.395,Z 853.667,A -85,B 0,C 180,E1 -9453.736,E2 -9453.736} C_VEL
LIN {X 0,Y 431.39,Z 850.663,A -85,B 0,C 180,E1 -9455.141,E2 -9455.141} C_VEL
LIN {X 0,Y 431.437,Z 846.584,A -85,B 0,C 180,E1 -9456.547,E2 -9456.547} C_VEL
LIN {X 0,Y 431.603,Z 840.293,A -85,B 0,C 180,E1 -9458.191,E2 -9458.191} C_VEL
LIN {X 0,Y 431.867,Z 833.437,A -85,B 0,C 180,E1 -9459.602,E2 -9459.602} C_VEL
LIN {X 0,Y 432.344,Z 824.928,A -85,B 0,C 180,E1 -9461.011,E2 -9461.011} C_VEL
LIN {X 0,Y 432.804,Z 816.153,A -85,B 0,C 180,E1 -9462.186,E2 -9462.186} C_VEL
LIN {X 0,Y 433.384,Z 806.211,A -85,B 0,C 180,E1 -9463.276,E2 -9463.276} C_VEL
LIN {X 0,Y 434.131,Z 794.666,A -85,B 0,C 180,E1 -9464.292,E2 -9464.292} C_VEL
LIN {X 0,Y 434.826,Z 782.732,A -85,B 0,C 180,E1 -9465.107,E2 -9465.107} C_VEL
LIN {X 0,Y 435.354,Z 770.345,A -85,B 0,C 180,E1 -9465.748,E2 -9465.748} C_VEL
LIN {X 0,Y 435.929,Z 757.7,A -85,B 0,C 180,E1 -9466.207,E2 -9466.207} C_VEL
LIN {X 0,Y 436.281,Z 742.902,A -85,B 0,C 180,E1 -9466.524,E2 -9466.524} C_VEL
LIN {X 0,Y 436.982,Z 667.245,A -85,B 0,C 180,E1 -9467.822,E2 -9467.822} C_VEL
LIN {X 0,Y 433.968,Z 641.865,A -85,B 0,C 180,E1 -9468.415,E2 -9468.415} C_VEL
LIN {X 0,Y 435.115,Z 619.743,A -85,B 0,C 180,E1 -9471.558,E2 -9471.558} C_VEL
LIN {X 0,Y 436.472,Z 597.535,A -85,B 0,C 180,E1 -9474.749,E2 -9474.749} C_VEL
LIN {X 0,Y 436.252,Z 593.837,A -85,B 0,C 180,E1 -9475.305,E2 -9475.305} C_VEL
LIN {X 0,Y 432.763,Z 578.192,A -85,B 0,C 180,E1 -9477.832,E2 -9477.832} C_VEL
LIN {X 0,Y 432.415,Z 576.623,A -85,B 0,C 180,E1 -9478.12,E2 -9478.12} C_VEL
LIN {X 0,Y 432.32,Z 576.634,A -85,B 0,C 180,E1 -9481.345,E2 -9481.345} C_VEL
LIN {X 0,Y 432.339,Z 576.629,A -85,B 0,C 180,E1 -9484.676,E2 -9484.676} C_VEL
LIN {X 0,Y 432.348,Z 576.628,A -85,B 0,C 180,E1 -9488.148,E2 -9488.148} C_VEL
LIN {X 0,Y 432.363,Z 576.625,A -85,B 0,C 180,E1 -9491.606,E2 -9491.606} C_VEL
LIN {X 0,Y 432.374,Z 576.623,A -85,B 0,C 180,E1 -9495.658,E2 -9495.658} C_VEL
LIN {X 0,Y 432.368,Z 576.627,A -85,B 0,C 180,E1 -9498.391,E2 -9498.391} C_VEL
LIN {X 0,Y 432.348,Z 576.626,A -85,B 0,C 180,E1 -9501.851,E2 -9501.851} C_VEL
LIN {X 0,Y 432.334,Z 576.619,A -85,B 0,C 180,E1 -9505.322,E2 -9505.322} C_VEL
LIN {X 0,Y 432.326,Z 576.631,A -85,B 0,C 180,E1 -9508.654,E2 -9508.654} C_VEL
LIN {X 0,Y 432.377,Z 576.615,A -85,B 0,C 180,E1 -9511.876,E2 -9511.876} C_VEL
LIN {X 0,Y 432.344,Z 576.626,A -85,B 0,C 180,E1 -9514.998,E2 -9514.998} C_VEL
LIN {X 0,Y 432.349,Z 576.617,A -85,B 0,C 180,E1 -9518.045,E2 -9518.045} C_VEL
LIN {X 0,Y 432.378,Z 576.623,A -85,B 0,C 180,E1 -9521.029,E2 -9521.029} C_VEL
LIN {X 0,Y 432.421,Z 576.609,A -85,B 0,C 180,E1 -9523.961,E2 -9523.961} C_VEL
LIN {X 0,Y 432.45,Z 576.614,A -85,B 0,C 180,E1 -9527.803,E2 -9527.803} C_VEL
LIN {X 0,Y 432.483,Z 576.598,A -85,B 0,C 180,E1 -9531.59,E2 -9531.59} C_VEL
LIN {X 0,Y 432.595,Z 576.599,A -85,B 0,C 180,E1 -9534.406,E2 -9534.406} C_VEL
LIN {X 0,Y 432.597,Z 576.587,A -85,B 0,C 180,E1 -9538.138,E2 -9538.138} C_VEL
LIN {X 0,Y 432.725,Z 576.574,A -85,B 0,C 180,E1 -9540,E2 -9540} C_VEL
LIN {X 0,Y 432.597,Z 576.6,A -85,B 0,C 180,E1 -9542.794,E2 -9542.794} C_VEL
LIN {X 0,Y 432.565,Z 576.591,A -85,B 0,C 180,E1 -9546.53,E2 -9546.53} C_VEL
LIN {X 0,Y 432.434,Z 576.617,A -85,B 0,C 180,E1 -9549.353,E2 -9549.353} C_VEL
LIN {X 0,Y 432.422,Z 576.611,A -85,B 0,C 180,E1 -9552.804,E2 -9552.804} C_VEL
LIN {X 0,Y 432.403,Z 576.622,A -85,B 0,C 180,E1 -9556.479,E2 -9556.479} C_VEL
LIN {X 0,Y 432.33,Z 576.624,A -85,B 0,C 180,E1 -9559.961,E2 -9559.961} C_VEL
LIN {X 0,Y 432.31,Z 576.634,A -85,B 0,C 180,E1 -9562.965,E2 -9562.965} C_VEL
LIN {X 0,Y 432.357,Z 576.623,A -85,B 0,C 180,E1 -9566.033,E2 -9566.033} C_VEL
LIN {X 0,Y 432.345,Z 576.625,A -85,B 0,C 180,E1 -9569.187,E2 -9569.187} C_VEL
LIN {X 0,Y 432.326,Z 576.63,A -85,B 0,C 180,E1 -9572.296,E2 -9572.296} C_VEL
LIN {X 0,Y 432.334,Z 576.625,A -85,B 0,C 180,E1 -9574.678,E2 -9574.678} C_VEL
LIN {X 0,Y 432.343,Z 576.627,A -85,B 0,C 180,E1 -9578.149,E2 -9578.149} C_VEL
LIN {X 0,Y 432.361,Z 576.609,A -85,B 0,C 180,E1 -9581.608,E2 -9581.608} C_VEL
LIN {X 0,Y 432.336,Z 576.627,A -85,B 0,C 180,E1 -9584.347,E2 -9584.347} C_VEL
LIN {X 0,Y 432.316,Z 576.627,A -85,B 0,C 180,E1 -9587.017,E2 -9587.017} C_VEL
LIN {X 0,Y 432.33,Z 576.632,A -85,B 0,C 180,E1 -9589.822,E2 -9589.822} C_VEL
LIN {X 0,Y 432.313,Z 576.63,A -85,B 0,C 180,E1 -9593.024,E2 -9593.024} C_VEL
LIN {X 0,Y 432.358,Z 576.628,A -85,B 0,C 180,E1 -9595.997,E2 -9595.997} C_VEL
LIN {X 0,Y 432.326,Z 576.67,A -85,B 0,C 180,E1 -9599.495,E2 -9599.495} C_VEL
LIN {X 0,Y 434.065,Z 581.32,A -85,B 0,C 180,E1 -9599.665,E2 -9599.665} C_VEL
LIN {X 0,Y 437.96,Z 590.897,A -85,B 0,C 180,E1 -9600.026,E2 -9600.026} C_VEL
LIN {X 0,Y 436.885,Z 678.877,A -85,B 0,C 180,E1 -9601.507,E2 -9601.507} C_VEL
LIN {X 0,Y 436.66,Z 692.148,A -85,B 0,C 180,E1 -9601.916,E2 -9601.916} C_VEL
LIN {X 0,Y 436.295,Z 704.502,A -85,B 0,C 180,E1 -9602.495,E2 -9602.495} C_VEL
LIN {X 0,Y 435.726,Z 716.967,A -85,B 0,C 180,E1 -9603.282,E2 -9603.282} C_VEL
LIN {X 0,Y 435.11,Z 727.559,A -85,B 0,C 180,E1 -9604.145,E2 -9604.145} C_VEL
LIN {X 0,Y 434.361,Z 738.329,A -85,B 0,C 180,E1 -9605.251,E2 -9605.251} C_VEL
LIN {X 0,Y 433.833,Z 747.086,A -85,B 0,C 180,E1 -9606.363,E2 -9606.363} C_VEL
LIN {X 0,Y 433.251,Z 755.179,A -85,B 0,C 180,E1 -9607.613,E2 -9607.613} C_VEL
LIN {X 0,Y 432.656,Z 762.728,A -85,B 0,C 180,E1 -9609.062,E2 -9609.062} C_VEL
LIN {X 0,Y 432.234,Z 768.964,A -85,B 0,C 180,E1 -9610.573,E2 -9610.573} C_VEL
LIN {X 0,Y 431.949,Z 773.538,A -85,B 0,C 180,E1 -9611.993,E2 -9611.993} C_VEL
LIN {X 0,Y 431.8,Z 776.031,A -85,B 0,C 180,E1 -9612.965,E2 -9612.965} C_VEL
LIN {X 0,Y 431.673,Z 778.012,A -85,B 0,C 180,E1 -9613.933,E2 -9613.933} C_VEL
LIN {X 0,Y 431.456,Z 780.354,A -85,B 0,C 180,E1 -9615.575,E2 -9615.575} C_VEL
LIN {X 0,Y 430.761,Z 781.167,A -85,B 0,C 180,E1 -9616.348,E2 -9616.348} C_VEL
LIN {X 0,Y 427.869,Z 782.027,A -85,B 0,C 180,E1 -9617.611,E2 -9617.611} C_VEL
LIN {X 0,Y 425.443,Z 782.118,A -85,B 0,C 180,E1 -9618.631,E2 -9618.631} C_VEL
LIN {X 0,Y 424.408,Z 781.75,A -85,B 0,C 180,E1 -9619.419,E2 -9619.419} C_VEL
LIN {X 0,Y 424.328,Z 781.529,A -85,B 0,C 180,E1 -9619.684,E2 -9619.684} C_VEL
LIN {X 0,Y 424.457,Z 779.521,A -85,B 0,C 180,E1 -9621.43,E2 -9621.43} C_VEL
LIN {X 0,Y 424.727,Z 776.205,A -85,B 0,C 180,E1 -9623.134,E2 -9623.134} C_VEL
LIN {X 0,Y 424.932,Z 771.582,A -85,B 0,C 180,E1 -9624.781,E2 -9624.781} C_VEL
LIN {X 0,Y 425.274,Z 765.372,A -85,B 0,C 180,E1 -9626.447,E2 -9626.447} C_VEL
LIN {X 0,Y 425.751,Z 758.557,A -85,B 0,C 180,E1 -9627.872,E2 -9627.872} C_VEL
LIN {X 0,Y 426.316,Z 750.06,A -85,B 0,C 180,E1 -9629.292,E2 -9629.292} C_VEL
LIN {X 0,Y 426.922,Z 741.369,A -85,B 0,C 180,E1 -9630.472,E2 -9630.472} C_VEL
LIN {X 0,Y 427.47,Z 731.86,A -85,B 0,C 180,E1 -9631.531,E2 -9631.531} C_VEL
LIN {X 0,Y 428.085,Z 721.359,A -85,B 0,C 180,E1 -9632.47,E2 -9632.47} C_VEL
LIN {X 0,Y 428.696,Z 709.738,A -85,B 0,C 180,E1 -9633.289,E2 -9633.289} C_VEL
LIN {X 0,Y 429.114,Z 697.815,A -85,B 0,C 180,E1 -9633.932,E2 -9633.932} C_VEL
LIN {X 0,Y 429.452,Z 685.502,A -85,B 0,C 180,E1 -9634.399,E2 -9634.399} C_VEL
LIN {X 0,Y 429.632,Z 671.752,A -85,B 0,C 180,E1 -9634.721,E2 -9634.721} C_VEL
LIN {X 0,Y 430.374,Z 591.727,A -85,B 0,C 180,E1 -9636.058,E2 -9636.058} C_VEL
LIN {X 0,Y 425.526,Z 577.481,A -85,B 0,C 180,E1 -9636.52,E2 -9636.52} C_VEL
LIN {X 0,Y 425.403,Z 577.494,A -85,B 0,C 180,E1 -9639.509,E2 -9639.509} C_VEL
LIN {X 0,Y 425.406,Z 577.491,A -85,B 0,C 180,E1 -9642.91,E2 -9642.91} C_VEL
LIN {X 0,Y 425.363,Z 577.499,A -85,B 0,C 180,E1 -9646.605,E2 -9646.605} C_VEL
LIN {X 0,Y 425.33,Z 577.504,A -85,B 0,C 180,E1 -9649.635,E2 -9649.635} C_VEL
LIN {X 0,Y 425.288,Z 577.509,A -85,B 0,C 180,E1 -9652.338,E2 -9652.338} C_VEL
LIN {X 0,Y 425.289,Z 577.508,A -85,B 0,C 180,E1 -9655.445,E2 -9655.445} C_VEL
LIN {X 0,Y 425.386,Z 577.597,A -85,B 0,C 180,E1 -9657.453,E2 -9657.453} C_VEL
LIN {X 0,Y 430.593,Z 591.906,A -85,B 0,C 180,E1 -9657.941,E2 -9657.941} C_VEL
LIN {X 0,Y 429.503,Z 679.534,A -85,B 0,C 180,E1 -9659.496,E2 -9659.496} C_VEL
LIN {X 0,Y 429.266,Z 693.082,A -85,B 0,C 180,E1 -9659.939,E2 -9659.939} C_VEL
LIN {X 0,Y 428.896,Z 705.363,A -85,B 0,C 180,E1 -9660.528,E2 -9660.528} C_VEL
LIN {X 0,Y 428.308,Z 717.686,A -85,B 0,C 180,E1 -9661.331,E2 -9661.331} C_VEL
LIN {X 0,Y 427.738,Z 728.933,A -85,B 0,C 180,E1 -9662.275,E2 -9662.275} C_VEL
LIN {X 0,Y 427.124,Z 738.975,A -85,B 0,C 180,E1 -9663.324,E2 -9663.324} C_VEL
LIN {X 0,Y 426.484,Z 748.218,A -85,B 0,C 180,E1 -9664.518,E2 -9664.518} C_VEL
LIN {X 0,Y 425.958,Z 756.535,A -85,B 0,C 180,E1 -9665.839,E2 -9665.839} C_VEL
LIN {X 0,Y 425.44,Z 763.79,A -85,B 0,C 180,E1 -9667.259,E2 -9667.259} C_VEL
LIN {X 0,Y 425.137,Z 769.331,A -85,B 0,C 180,E1 -9668.611,E2 -9668.611} C_VEL
LIN {X 0,Y 424.758,Z 774.411,A -85,B 0,C 180,E1 -9670.186,E2 -9670.186} C_VEL
LIN {X 0,Y 424.551,Z 778.297,A -85,B 0,C 180,E1 -9671.847,E2 -9671.847} C_VEL
LIN {X 0,Y 424.398,Z 780.542,A -85,B 0,C 180,E1 -9673.228,E2 -9673.228} C_VEL
LIN {X 0,Y 424.316,Z 781.911,A -85,B 0,C 180,E1 -9674.584,E2 -9674.584} C_VEL
LIN {X 0,Y 424.29,Z 782.435,A -85,B 0,C 180,E1 -9675.917,E2 -9675.917} C_VEL
LIN {X 0,Y 424.297,Z 782.192,A -85,B 0,C 180,E1 -9677.225,E2 -9677.225} C_VEL
LIN {X 0,Y 424.401,Z 781.229,A -85,B 0,C 180,E1 -9678.517,E2 -9678.517} C_VEL
LIN {X 0,Y 424.605,Z 778.436,A -85,B 0,C 180,E1 -9680.413,E2 -9680.413} C_VEL
LIN {X 0,Y 424.93,Z 774.011,A -85,B 0,C 180,E1 -9682.269,E2 -9682.269} C_VEL
LIN {X 0,Y 425.321,Z 767.999,A -85,B 0,C 180,E1 -9684.062,E2 -9684.062} C_VEL
LIN {X 0,Y 425.792,Z 761.108,A -85,B 0,C 180,E1 -9685.615,E2 -9685.615} C_VEL
LIN {X 0,Y 426.389,Z 753.089,A -85,B 0,C 180,E1 -9687.049,E2 -9687.049} C_VEL
LIN {X 0,Y 426.981,Z 745.057,A -85,B 0,C 180,E1 -9688.216,E2 -9688.216} C_VEL
LIN {X 0,Y 427.646,Z 735.343,A -85,B 0,C 180,E1 -9689.372,E2 -9689.372} C_VEL
LIN {X 0,Y 428.298,Z 724.305,A -85,B 0,C 180,E1 -9690.419,E2 -9690.419} C_VEL
LIN {X 0,Y 428.9,Z 712.627,A -85,B 0,C 180,E1 -9691.294,E2 -9691.294} C_VEL
LIN {X 0,Y 429.395,Z 701.411,A -85,B 0,C 180,E1 -9691.937,E2 -9691.937} C_VEL
LIN {X 0,Y 429.706,Z 688.517,A -85,B 0,C 180,E1 -9692.474,E2 -9692.474} C_VEL
LIN {X 0,Y 429.916,Z 674.869,A -85,B 0,C 180,E1 -9692.832,E2 -9692.832} C_VEL
LIN {X 0,Y 431.015,Z 592.1,A -85,B 0,C 180,E1 -9694.302,E2 -9694.302} C_VEL
LIN {X 0,Y 425.483,Z 578.202,A -85,B 0,C 180,E1 -9694.842,E2 -9694.842} C_VEL
LIN {X 0,Y 425.348,Z 577.503,A -85,B 0,C 180,E1 -9694.889,E2 -9694.889} C_VEL
LIN {X 0,Y 425.284,Z 577.511,A -85,B 0,C 180,E1 -9697.729,E2 -9697.729} C_VEL
LIN {X 0,Y 425.353,Z 577.503,A -85,B 0,C 180,E1 -9700.704,E2 -9700.704} C_VEL
LIN {X 0,Y 425.379,Z 577.496,A -85,B 0,C 180,E1 -9703.688,E2 -9703.688} C_VEL
LIN {X 0,Y 425.423,Z 577.491,A -85,B 0,C 180,E1 -9707.598,E2 -9707.598} C_VEL
LIN {X 0,Y 425.434,Z 577.489,A -85,B 0,C 180,E1 -9711.45,E2 -9711.45} C_VEL
LIN {X 0,Y 425.569,Z 577.477,A -85,B 0,C 180,E1 -9714.313,E2 -9714.313} C_VEL
LIN {X 0,Y 425.566,Z 577.472,A -85,B 0,C 180,E1 -9718.107,E2 -9718.107} C_VEL
LIN {X 0,Y 425.695,Z 577.458,A -85,B 0,C 180,E1 -9720,E2 -9720} C_VEL
LIN {X 0,Y 425.549,Z 577.474,A -85,B 0,C 180,E1 -9722.84,E2 -9722.84} C_VEL
LIN {X 0,Y 425.57,Z 577.471,A -85,B 0,C 180,E1 -9725.687,E2 -9725.687} C_VEL
LIN {X 0,Y 425.434,Z 577.492,A -85,B 0,C 180,E1 -9728.55,E2 -9728.55} C_VEL
LIN {X 0,Y 425.421,Z 577.492,A -85,B 0,C 180,E1 -9732.402,E2 -9732.402} C_VEL
LIN {X 0,Y 425.379,Z 577.495,A -85,B 0,C 180,E1 -9736.312,E2 -9736.312} C_VEL
LIN {X 0,Y 425.32,Z 577.499,A -85,B 0,C 180,E1 -9739.636,E2 -9739.636} C_VEL
LIN {X 0,Y 425.3,Z 577.501,A -85,B 0,C 180,E1 -9743.366,E2 -9743.366} C_VEL
LIN {X 0,Y 425.341,Z 577.498,A -85,B 0,C 180,E1 -9746.845,E2 -9746.845} C_VEL
LIN {X 0,Y 425.311,Z 577.504,A -85,B 0,C 180,E1 -9749.718,E2 -9749.718} C_VEL
LIN {X 0,Y 425.276,Z 577.507,A -85,B 0,C 180,E1 -9753.049,E2 -9753.049} C_VEL
LIN {X 0,Y 425.279,Z 577.509,A -85,B 0,C 180,E1 -9755.93,E2 -9755.93} C_VEL
LIN {X 0,Y 425.308,Z 577.504,A -85,B 0,C 180,E1 -9759.047,E2 -9759.047} C_VEL
LIN {X 0,Y 425.327,Z 577.507,A -85,B 0,C 180,E1 -9762.647,E2 -9762.647} C_VEL
LIN {X 0,Y 425.29,Z 577.508,A -85,B 0,C 180,E1 -9765.283,E2 -9765.283} C_VEL
LIN {X 0,Y 425.301,Z 577.511,A -85,B 0,C 180,E1 -9768.626,E2 -9768.626} C_VEL
LIN {X 0,Y 425.32,Z 577.505,A -85,B 0,C 180,E1 -9771.105,E2 -9771.105} C_VEL
LIN {X 0,Y 425.298,Z 577.509,A -85,B 0,C 180,E1 -9774.665,E2 -9774.665} C_VEL
LIN {X 0,Y 425.264,Z 577.516,A -85,B 0,C 180,E1 -9778.074,E2 -9778.074} C_VEL
LIN {X 0,Y 425.325,Z 577.571,A -85,B 0,C 180,E1 -9780.113,E2 -9780.113} C_VEL
LIN {X 0,Y 428.196,Z 590.557,A -85,B 0,C 180,E1 -9782.642,E2 -9782.642} C_VEL
LIN {X 0,Y 429.117,Z 596.569,A -85,B 0,C 180,E1 -9783.756,E2 -9783.756} C_VEL
LIN {X 0,Y 427.946,Z 614.915,A -85,B 0,C 180,E1 -9786.878,E2 -9786.878} C_VEL
LIN {X 0,Y 426.817,Z 635.195,A -85,B 0,C 180,E1 -9790.273,E2 -9790.273} C_VEL
LIN {X 0,Y 426.512,Z 640.62,A -85,B 0,C 180,E1 -9791.153,E2 -9791.153} C_VEL
LIN {X 0,Y 430.336,Z 669.778,A -85,B 0,C 180,E1 -9791.869,E2 -9791.869} C_VEL
LIN {X 0,Y 429.375,Z 751.18,A -85,B 0,C 180,E1 -9793.325,E2 -9793.325} C_VEL
LIN {X 0,Y 428.873,Z 764.875,A -85,B 0,C 180,E1 -9793.764,E2 -9793.764} C_VEL
LIN {X 0,Y 428.187,Z 777.309,A -85,B 0,C 180,E1 -9794.348,E2 -9794.348} C_VEL
LIN {X 0,Y 427.474,Z 789.289,A -85,B 0,C 180,E1 -9795.115,E2 -9795.115} C_VEL
LIN {X 0,Y 426.776,Z 800.773,A -85,B 0,C 180,E1 -9796.058,E2 -9796.058} C_VEL
LIN {X 0,Y 426.199,Z 811.301,A -85,B 0,C 180,E1 -9797.138,E2 -9797.138} C_VEL
LIN {X 0,Y 425.602,Z 818.966,A -85,B 0,C 180,E1 -9798.088,E2 -9798.088} C_VEL
LIN {X 0,Y 425.092,Z 827.058,A -85,B 0,C 180,E1 -9799.281,E2 -9799.281} C_VEL
LIN {X 0,Y 424.704,Z 834.996,A -85,B 0,C 180,E1 -9800.715,E2 -9800.715} C_VEL
LIN {X 0,Y 424.44,Z 842.326,A -85,B 0,C 180,E1 -9802.388,E2 -9802.388} C_VEL
LIN {X 0,Y 424.292,Z 847.564,A -85,B 0,C 180,E1 -9803.931,E2 -9803.931} C_VEL
LIN {X 0,Y 424.262,Z 850.974,A -85,B 0,C 180,E1 -9805.249,E2 -9805.249} C_VEL
LIN {X 0,Y 424.29,Z 852.918,A -85,B 0,C 180,E1 -9806.201,E2 -9806.201} C_VEL
LIN {X 0,Y 424.356,Z 854.382,A -85,B 0,C 180,E1 -9807.152,E2 -9807.152} C_VEL
LIN {X 0,Y 424.357,Z 855.431,A -85,B 0,C 180,E1 -9808.102,E2 -9808.102} C_VEL
LIN {X 0,Y 424.265,Z 856.072,A -85,B 0,C 180,E1 -9809.051,E2 -9809.051} C_VEL
LIN {X 0,Y 424.24,Z 856.304,A -85,B 0,C 180,E1 -9810,E2 -9810} C_VEL
LIN {X 0,Y 424.357,Z 855.492,A -85,B 0,C 180,E1 -9811.898,E2 -9811.898} C_VEL
LIN {X 0,Y 424.356,Z 854.48,A -85,B 0,C 180,E1 -9812.848,E2 -9812.848} C_VEL
LIN {X 0,Y 424.301,Z 853.031,A -85,B 0,C 180,E1 -9813.799,E2 -9813.799} C_VEL
LIN {X 0,Y 424.325,Z 850.022,A -85,B 0,C 180,E1 -9815.226,E2 -9815.226} C_VEL
LIN {X 0,Y 424.349,Z 845.929,A -85,B 0,C 180,E1 -9816.657,E2 -9816.657} C_VEL
LIN {X 0,Y 424.53,Z 839.622,A -85,B 0,C 180,E1 -9818.329,E2 -9818.329} C_VEL
LIN {X 0,Y 424.83,Z 832.752,A -85,B 0,C 180,E1 -9819.762,E2 -9819.762} C_VEL
LIN {X 0,Y 425.331,Z 824.216,A -85,B 0,C 180,E1 -9821.195,E2 -9821.195} C_VEL
LIN {X 0,Y 425.811,Z 815.414,A -85,B 0,C 180,E1 -9822.39,E2 -9822.39} C_VEL
LIN {X 0,Y 426.355,Z 805.872,A -85,B 0,C 180,E1 -9823.454,E2 -9823.454} C_VEL
LIN {X 0,Y 427.116,Z 795.301,A -85,B 0,C 180,E1 -9824.411,E2 -9824.411} C_VEL
LIN {X 0,Y 427.801,Z 783.814,A -85,B 0,C 180,E1 -9825.239,E2 -9825.239} C_VEL
LIN {X 0,Y 428.371,Z 771.975,A -85,B 0,C 180,E1 -9825.889,E2 -9825.889} C_VEL
LIN {X 0,Y 429.022,Z 758.413,A -85,B 0,C 180,E1 -9826.414,E2 -9826.414} C_VEL
LIN {X 0,Y 429.382,Z 744.812,A -85,B 0,C 180,E1 -9826.736,E2 -9826.736} C_VEL
LIN {X 0,Y 430.145,Z 667.676,A -85,B 0,C 180,E1 -9828.085,E2 -9828.085} C_VEL
LIN {X 0,Y 427.031,Z 641.346,A -85,B 0,C 180,E1 -9828.705,E2 -9828.705} C_VEL
LIN {X 0,Y 428.15,Z 620.802,A -85,B 0,C 180,E1 -9831.674,E2 -9831.674} C_VEL
LIN {X 0,Y 429.564,Z 598.58,A -85,B 0,C 180,E1 -9834.915,E2 -9834.915} C_VEL
LIN {X 0,Y 429.22,Z 594.716,A -85,B 0,C 180,E1 -9835.513,E2 -9835.513} C_VEL
LIN {X 0,Y 425.757,Z 579.226,A -85,B 0,C 180,E1 -9838.063,E2 -9838.063} C_VEL
LIN {X 0,Y 425.368,Z 577.5,A -85,B 0,C 180,E1 -9838.359,E2 -9838.359} C_VEL
LIN {X 0,Y 425.264,Z 577.515,A -85,B 0,C 180,E1 -9841.926,E2 -9841.926} C_VEL
LIN {X 0,Y 425.299,Z 577.506,A -85,B 0,C 180,E1 -9845.335,E2 -9845.335} C_VEL
LIN {X 0,Y 425.308,Z 577.502,A -85,B 0,C 180,E1 -9849.045,E2 -9849.045} C_VEL
LIN {X 0,Y 425.312,Z 577.503,A -85,B 0,C 180,E1 -9851.961,E2 -9851.961} C_VEL
LIN {X 0,Y 425.309,Z 577.501,A -85,B 0,C 180,E1 -9855.278,E2 -9855.278} C_VEL
LIN {X 0,Y 425.305,Z 577.504,A -85,B 0,C 180,E1 -9858.625,E2 -9858.625} C_VEL
LIN {X 0,Y 425.319,Z 577.499,A -85,B 0,C 180,E1 -9861.103,E2 -9861.103} C_VEL
LIN {X 0,Y 425.294,Z 577.499,A -85,B 0,C 180,E1 -9864.663,E2 -9864.663} C_VEL
LIN {X 0,Y 425.267,Z 577.512,A -85,B 0,C 180,E1 -9868.073,E2 -9868.073} C_VEL
LIN {X 0,Y 425.331,Z 577.491,A -85,B 0,C 180,E1 -9871.368,E2 -9871.368} C_VEL
LIN {X 0,Y 425.288,Z 577.51,A -85,B 0,C 180,E1 -9874.554,E2 -9874.554} C_VEL
LIN {X 0,Y 425.279,Z 577.495,A -85,B 0,C 180,E1 -9877.661,E2 -9877.661} C_VEL
LIN {X 0,Y 425.353,Z 577.502,A -85,B 0,C 180,E1 -9880.704,E2 -9880.704} C_VEL
LIN {X 0,Y 425.379,Z 577.485,A -85,B 0,C 180,E1 -9883.688,E2 -9883.688} C_VEL
LIN {X 0,Y 425.403,Z 577.491,A -85,B 0,C 180,E1 -9887.598,E2 -9887.598} C_VEL
LIN {X 0,Y 425.433,Z 577.476,A -85,B 0,C 180,E1 -9891.45,E2 -9891.45} C_VEL
LIN {X 0,Y 425.57,Z 577.473,A -85,B 0,C 180,E1 -9894.313,E2 -9894.313} C_VEL
LIN {X 0,Y 425.567,Z 577.463,A -85,B 0,C 180,E1 -9898.107,E2 -9898.107} C_VEL
LIN {X 0,Y 425.695,Z 577.449,A -85,B 0,C 180,E1 -9900,E2 -9900} C_VEL
LIN {X 0,Y 425.549,Z 577.477,A -85,B 0,C 180,E1 -9902.84,E2 -9902.84} C_VEL
LIN {X 0,Y 425.522,Z 577.469,A -85,B 0,C 180,E1 -9906.639,E2 -9906.639} C_VEL
LIN {X 0,Y 425.393,Z 577.493,A -85,B 0,C 180,E1 -9909.51,E2 -9909.51} C_VEL
LIN {X 0,Y 425.384,Z 577.488,A -85,B 0,C 180,E1 -9912.904,E2 -9912.904} C_VEL
LIN {X 0,Y 425.352,Z 577.502,A -85,B 0,C 180,E1 -9916.605,E2 -9916.605} C_VEL
LIN {X 0,Y 425.32,Z 577.498,A -85,B 0,C 180,E1 -9919.636,E2 -9919.636} C_VEL
LIN {X 0,Y 425.279,Z 577.508,A -85,B 0,C 180,E1 -9922.339,E2 -9922.339} C_VEL
LIN {X 0,Y 425.288,Z 577.506,A -85,B 0,C 180,E1 -9925.446,E2 -9925.446} C_VEL
LIN {X 0,Y 425.331,Z 577.503,A -85,B 0,C 180,E1 -9928.632,E2 -9928.632} C_VEL
LIN {X 0,Y 425.268,Z 577.509,A -85,B 0,C 180,E1 -9931.927,E2 -9931.927} C_VEL
LIN {X 0,Y 425.294,Z 577.508,A -85,B 0,C 180,E1 -9935.337,E2 -9935.337} C_VEL
LIN {X 0,Y 425.302,Z 577.51,A -85,B 0,C 180,E1 -9939.046,E2 -9939.046} C_VEL
LIN {X 0,Y 425.311,Z 577.485,A -85,B 0,C 180,E1 -9941.963,E2 -9941.963} C_VEL
LIN {X 0,Y 425.282,Z 577.513,A -85,B 0,C 180,E1 -9945.284,E2 -9945.284} C_VEL
LIN {X 0,Y 425.27,Z 577.502,A -85,B 0,C 180,E1 -9948.622,E2 -9948.622} C_VEL
LIN {X 0,Y 425.309,Z 577.504,A -85,B 0,C 180,E1 -9951.104,E2 -9951.104} C_VEL
LIN {X 0,Y 425.299,Z 577.506,A -85,B 0,C 180,E1 -9954.665,E2 -9954.665} C_VEL
LIN {X 0,Y 425.264,Z 577.511,A -85,B 0,C 180,E1 -9958.074,E2 -9958.074} C_VEL
LIN {X 0,Y 425.314,Z 577.665,A -85,B 0,C 180,E1 -9959.145,E2 -9959.145} C_VEL
LIN {X 0,Y 428.986,Z 586.777,A -85,B 0,C 180,E1 -9959.5,E2 -9959.5} C_VEL
LIN {X 0,Y 431.322,Z 592.563,A -85,B 0,C 180,E1 -9959.722,E2 -9959.722} C_VEL
LIN {X 0,Y 430.179,Z 680.044,A -85,B 0,C 180,E1 -9961.221,E2 -9961.221} C_VEL
LIN {X 0,Y 429.963,Z 693.103,A -85,B 0,C 180,E1 -9961.639,E2 -9961.639} C_VEL
LIN {X 0,Y 429.575,Z 704.985,A -85,B 0,C 180,E1 -9962.205,E2 -9962.205} C_VEL
LIN {X 0,Y 429.017,Z 716.869,A -85,B 0,C 180,E1 -9962.962,E2 -9962.962} C_VEL
LIN {X 0,Y 428.359,Z 727.61,A -85,B 0,C 180,E1 -9963.837,E2 -9963.837} C_VEL
LIN {X 0,Y 427.563,Z 738.489,A -85,B 0,C 180,E1 -9964.96,E2 -9964.96} C_VEL
LIN {X 0,Y 426.92,Z 748.206,A -85,B 0,C 180,E1 -9966.215,E2 -9966.215} C_VEL
LIN {X 0,Y 426.326,Z 755.681,A -85,B 0,C 180,E1 -9967.393,E2 -9967.393} C_VEL
LIN {X 0,Y 425.683,Z 763.658,A -85,B 0,C 180,E1 -9968.956,E2 -9968.956} C_VEL
LIN {X 0,Y 425.251,Z 769.479,A -85,B 0,C 180,E1 -9970.394,E2 -9970.394} C_VEL
LIN {X 0,Y 424.959,Z 773.642,A -85,B 0,C 180,E1 -9971.687,E2 -9971.687} C_VEL
LIN {X 0,Y 424.724,Z 777.317,A -85,B 0,C 180,E1 -9973.168,E2 -9973.168} C_VEL
LIN {X 0,Y 424.491,Z 779.922,A -85,B 0,C 180,E1 -9974.639,E2 -9974.639} C_VEL
LIN {X 0,Y 424.407,Z 781.123,A -85,B 0,C 180,E1 -9975.618,E2 -9975.618} C_VEL
LIN {X 0,Y 424.332,Z 781.874,A -85,B 0,C 180,E1 -9976.593,E2 -9976.593} C_VEL
LIN {X 0,Y 424.35,Z 782.229,A -85,B 0,C 180,E1 -9977.728,E2 -9977.728} C_VEL
LIN {X 0,Y 424.329,Z 781.697,A -85,B 0,C 180,E1 -9979.503,E2 -9979.503} C_VEL
LIN {X 0,Y 424.328,Z 781.529,A -85,B 0,C 180,E1 -9979.684,E2 -9979.684} C_VEL
LIN {X 0,Y 423.702,Z 780.871,A -85,B 0,C 180,E1 -9980.472,E2 -9980.472} C_VEL
LIN {X 0,Y 420.995,Z 779.336,A -85,B 0,C 180,E1 -9981.752,E2 -9981.752} C_VEL
LIN {X 0,Y 418.724,Z 777.661,A -85,B 0,C 180,E1 -9982.769,E2 -9982.769} C_VEL
LIN {X 0,Y 417.775,Z 775.958,A -85,B 0,C 180,E1 -9983.537,E2 -9983.537} C_VEL
LIN {X 0,Y 417.711,Z 775.291,A -85,B 0,C 180,E1 -9983.792,E2 -9983.792} C_VEL
LIN {X 0,Y 417.947,Z 771.166,A -85,B 0,C 180,E1 -9985.177,E2 -9985.177} C_VEL
LIN {X 0,Y 418.362,Z 764.599,A -85,B 0,C 180,E1 -9986.87,E2 -9986.87} C_VEL
LIN {X 0,Y 418.854,Z 757.455,A -85,B 0,C 180,E1 -9988.317,E2 -9988.317} C_VEL
LIN {X 0,Y 419.369,Z 750.178,A -85,B 0,C 180,E1 -9989.52,E2 -9989.52} C_VEL
LIN {X 0,Y 420.012,Z 741.382,A -85,B 0,C 180,E1 -9990.719,E2 -9990.719} C_VEL
LIN {X 0,Y 420.638,Z 730.471,A -85,B 0,C 180,E1 -9991.915,E2 -9991.915} C_VEL
LIN {X 0,Y 421.327,Z 719.508,A -85,B 0,C 180,E1 -9992.868,E2 -9992.868} C_VEL
LIN {X 0,Y 421.949,Z 707.108,A -85,B 0,C 180,E1 -9993.7,E2 -9993.7} C_VEL
LIN {X 0,Y 422.366,Z 694.586,A -85,B 0,C 180,E1 -9994.324,E2 -9994.324} C_VEL
LIN {X 0,Y 422.67,Z 682.543,A -85,B 0,C 180,E1 -9994.739,E2 -9994.739} C_VEL
LIN {X 0,Y 422.898,Z 662.491,A -85,B 0,C 180,E1 -9995.125,E2 -9995.125} C_VEL
LIN {X 0,Y 423.559,Z 593.122,A -85,B 0,C 180,E1 -9996.303,E2 -9996.303} C_VEL
LIN {X 0,Y 418.482,Z 578.357,A -85,B 0,C 180,E1 -9996.793,E2 -9996.793} C_VEL
LIN {X 0,Y 418.344,Z 578.374,A -85,B 0,C 180,E1 -9999.671,E2 -9999.671} C_VEL
LIN {X 0,Y 418.358,Z 578.369,A -85,B 0,C 180,E1 -10003.006,E2 -10003.006} C_VEL
LIN {X 0,Y 418.315,Z 578.376,A -85,B 0,C 180,E1 -10006.735,E2 -10006.735} C_VEL
LIN {X 0,Y 418.272,Z 578.384,A -85,B 0,C 180,E1 -10009.79,E2 -10009.79} C_VEL
LIN {X 0,Y 418.232,Z 578.385,A -85,B 0,C 180,E1 -10012.736,E2 -10012.736} C_VEL
LIN {X 0,Y 418.264,Z 578.388,A -85,B 0,C 180,E1 -10015.904,E2 -10015.904} C_VEL
LIN {X 0,Y 418.337,Z 578.424,A -85,B 0,C 180,E1 -10017.155,E2 -10017.155} C_VEL
LIN {X 0,Y 423.95,Z 593.878,A -85,B 0,C 180,E1 -10017.693,E2 -10017.693} C_VEL
LIN {X 0,Y 422.689,Z 679.746,A -85,B 0,C 180,E1 -10019.236,E2 -10019.236} C_VEL
LIN {X 0,Y 422.458,Z 693.266,A -85,B 0,C 180,E1 -10019.681,E2 -10019.681} C_VEL
LIN {X 0,Y 422.097,Z 705.024,A -85,B 0,C 180,E1 -10020.246,E2 -10020.246} C_VEL
LIN {X 0,Y 421.54,Z 716.555,A -85,B 0,C 180,E1 -10020.981,E2 -10020.981} C_VEL
LIN {X 0,Y 420.929,Z 728.123,A -85,B 0,C 180,E1 -10021.94,E2 -10021.94} C_VEL
LIN {X 0,Y 420.239,Z 738.675,A -85,B 0,C 180,E1 -10023.033,E2 -10023.033} C_VEL
LIN {X 0,Y 419.571,Z 748.339,A -85,B 0,C 180,E1 -10024.279,E2 -10024.279} C_VEL
LIN {X 0,Y 418.984,Z 756.917,A -85,B 0,C 180,E1 -10025.653,E2 -10025.653} C_VEL
LIN {X 0,Y 418.404,Z 764.724,A -85,B 0,C 180,E1 -10027.206,E2 -10027.206} C_VEL
LIN {X 0,Y 417.993,Z 771.26,A -85,B 0,C 180,E1 -10028.89,E2 -10028.89} C_VEL
LIN {X 0,Y 417.702,Z 775.396,A -85,B 0,C 180,E1 -10030.256,E2 -10030.256} C_VEL
LIN {X 0,Y 417.52,Z 778.555,A -85,B 0,C 180,E1 -10031.608,E2 -10031.608} C_VEL
LIN {X 0,Y 417.422,Z 779.891,A -85,B 0,C 180,E1 -10032.334,E2 -10032.334} C_VEL
LIN {X 0,Y 417.293,Z 781.72,A -85,B 0,C 180,E1 -10033.67,E2 -10033.67} C_VEL
LIN {X 0,Y 417.23,Z 782.771,A -85,B 0,C 180,E1 -10035.028,E2 -10035.028} C_VEL
LIN {X 0,Y 417.218,Z 783.048,A -85,B 0,C 180,E1 -10036.412,E2 -10036.412} C_VEL
LIN {X 0,Y 417.284,Z 782.5,A -85,B 0,C 180,E1 -10037.82,E2 -10037.82} C_VEL
LIN {X 0,Y 417.384,Z 781.06,A -85,B 0,C 180,E1 -10039.262,E2 -10039.262} C_VEL
LIN {X 0,Y 417.598,Z 778.642,A -85,B 0,C 180,E1 -10040.727,E2 -10040.727} C_VEL
LIN {X 0,Y 417.888,Z 775.109,A -85,B 0,C 180,E1 -10042.225,E2 -10042.225} C_VEL
LIN {X 0,Y 418.262,Z 769.484,A -85,B 0,C 180,E1 -10043.978,E2 -10043.978} C_VEL
LIN {X 0,Y 418.767,Z 762.652,A -85,B 0,C 180,E1 -10045.605,E2 -10045.605} C_VEL
LIN {X 0,Y 419.349,Z 755.071,A -85,B 0,C 180,E1 -10047.022,E2 -10047.022} C_VEL
LIN {X 0,Y 420.067,Z 746.047,A -85,B 0,C 180,E1 -10048.381,E2 -10048.381} C_VEL
LIN {X 0,Y 420.735,Z 736.824,A -85,B 0,C 180,E1 -10049.51,E2 -10049.51} C_VEL
LIN {X 0,Y 421.399,Z 726.529,A -85,B 0,C 180,E1 -10050.531,E2 -10050.531} C_VEL
LIN {X 0,Y 422.023,Z 715.042,A -85,B 0,C 180,E1 -10051.433,E2 -10051.433} C_VEL
LIN {X 0,Y 422.603,Z 702.605,A -85,B 0,C 180,E1 -10052.182,E2 -10052.182} C_VEL
LIN {X 0,Y 422.922,Z 689.684,A -85,B 0,C 180,E1 -10052.74,E2 -10052.74} C_VEL
LIN {X 0,Y 423.188,Z 676.061,A -85,B 0,C 180,E1 -10053.109,E2 -10053.109} C_VEL
LIN {X 0,Y 424.369,Z 594.184,A -85,B 0,C 180,E1 -10054.594,E2 -10054.594} C_VEL
LIN {X 0,Y 418.94,Z 580.492,A -85,B 0,C 180,E1 -10055.138,E2 -10055.138} C_VEL
LIN {X 0,Y 418.316,Z 578.378,A -85,B 0,C 180,E1 -10055.23,E2 -10055.23} C_VEL
LIN {X 0,Y 418.226,Z 578.389,A -85,B 0,C 180,E1 -10058.303,E2 -10058.303} C_VEL
LIN {X 0,Y 418.275,Z 578.382,A -85,B 0,C 180,E1 -10061.383,E2 -10061.383} C_VEL
LIN {X 0,Y 418.294,Z 578.384,A -85,B 0,C 180,E1 -10064.406,E2 -10064.406} C_VEL
LIN {X 0,Y 418.362,Z 578.371,A -85,B 0,C 180,E1 -10067.386,E2 -10067.386} C_VEL
LIN {X 0,Y 418.352,Z 578.374,A -85,B 0,C 180,E1 -10070.329,E2 -10070.329} C_VEL
LIN {X 0,Y 418.486,Z 578.355,A -85,B 0,C 180,E1 -10073.249,E2 -10073.249} C_VEL
LIN {X 0,Y 418.338,Z 578.373,A -85,B 0,C 180,E1 -10075.182,E2 -10075.182} C_VEL
LIN {X 0,Y 418.536,Z 578.347,A -85,B 0,C 180,E1 -10078.075,E2 -10078.075} C_VEL
LIN {X 0,Y 418.664,Z 578.333,A -85,B 0,C 180,E1 -10080,E2 -10080} C_VEL
LIN {X 0,Y 418.503,Z 578.351,A -85,B 0,C 180,E1 -10082.888,E2 -10082.888} C_VEL
LIN {X 0,Y 418.525,Z 578.349,A -85,B 0,C 180,E1 -10085.783,E2 -10085.783} C_VEL
LIN {X 0,Y 418.392,Z 578.367,A -85,B 0,C 180,E1 -10088.695,E2 -10088.695} C_VEL
LIN {X 0,Y 418.323,Z 578.37,A -85,B 0,C 180,E1 -10091.631,E2 -10091.631} C_VEL
LIN {X 0,Y 418.298,Z 578.377,A -85,B 0,C 180,E1 -10094.597,E2 -10094.597} C_VEL
LIN {X 0,Y 418.279,Z 578.373,A -85,B 0,C 180,E1 -10097.604,E2 -10097.604} C_VEL
LIN {X 0,Y 418.244,Z 578.382,A -85,B 0,C 180,E1 -10100.663,E2 -10100.663} C_VEL
LIN {X 0,Y 418.281,Z 578.376,A -85,B 0,C 180,E1 -10103.782,E2 -10103.782} C_VEL
LIN {X 0,Y 418.303,Z 578.373,A -85,B 0,C 180,E1 -10107.071,E2 -10107.071} C_VEL
LIN {X 0,Y 418.254,Z 578.385,A -85,B 0,C 180,E1 -10110.271,E2 -10110.271} C_VEL
LIN {X 0,Y 418.242,Z 578.382,A -85,B 0,C 180,E1 -10113.678,E2 -10113.678} C_VEL
LIN {X 0,Y 418.242,Z 578.385,A -85,B 0,C 180,E1 -10117.224,E2 -10117.224} C_VEL
LIN {X 0,Y 418.262,Z 578.38,A -85,B 0,C 180,E1 -10119.681,E2 -10119.681} C_VEL
LIN {X 0,Y 418.28,Z 578.382,A -85,B 0,C 180,E1 -10122.33,E2 -10122.33} C_VEL
LIN {X 0,Y 418.247,Z 578.386,A -85,B 0,C 180,E1 -10125.112,E2 -10125.112} C_VEL
LIN {X 0,Y 418.253,Z 578.385,A -85,B 0,C 180,E1 -10127.77,E2 -10127.77} C_VEL
LIN {X 0,Y 418.265,Z 578.386,A -85,B 0,C 180,E1 -10130.618,E2 -10130.618} C_VEL
LIN {X 0,Y 418.243,Z 578.387,A -85,B 0,C 180,E1 -10133.977,E2 -10133.977} C_VEL
LIN {X 0,Y 418.256,Z 578.385,A -85,B 0,C 180,E1 -10137.157,E2 -10137.157} C_VEL
LIN {X 0,Y 418.295,Z 578.452,A -85,B 0,C 180,E1 -10139.798,E2 -10139.798} C_VEL
LIN {X 0,Y 421.499,Z 593.11,A -85,B 0,C 180,E1 -10142.711,E2 -10142.711} C_VEL
LIN {X 0,Y 422.184,Z 597.52,A -85,B 0,C 180,E1 -10143.542,E2 -10143.542} C_VEL
LIN {X 0,Y 421.359,Z 610.932,A -85,B 0,C 180,E1 -10145.881,E2 -10145.881} C_VEL
LIN {X 0,Y 420.031,Z 632.417,A -85,B 0,C 180,E1 -10149.554,E2 -10149.554} C_VEL
LIN {X 0,Y 419.601,Z 639.753,A -85,B 0,C 180,E1 -10150.795,E2 -10150.795} C_VEL
LIN {X 0,Y 423.631,Z 670.871,A -85,B 0,C 180,E1 -10151.586,E2 -10151.586} C_VEL
LIN {X 0,Y 422.59,Z 750.865,A -85,B 0,C 180,E1 -10153.049,E2 -10153.049} C_VEL
LIN {X 0,Y 422.061,Z 764.435,A -85,B 0,C 180,E1 -10153.494,E2 -10153.494} C_VEL
LIN {X 0,Y 421.343,Z 776.798,A -85,B 0,C 180,E1 -10154.087,E2 -10154.087} C_VEL
LIN {X 0,Y 420.597,Z 788.743,A -85,B 0,C 180,E1 -10154.866,E2 -10154.866} C_VEL
LIN {X 0,Y 419.811,Z 800.67,A -85,B 0,C 180,E1 -10155.865,E2 -10155.865} C_VEL
LIN {X 0,Y 419.253,Z 810.724,A -85,B 0,C 180,E1 -10156.921,E2 -10156.921} C_VEL
LIN {X 0,Y 418.503,Z 820.115,A -85,B 0,C 180,E1 -10158.129,E2 -10158.129} C_VEL
LIN {X 0,Y 417.884,Z 829.284,A -85,B 0,C 180,E1 -10159.584,E2 -10159.584} C_VEL
LIN {X 0,Y 417.538,Z 836.7,A -85,B 0,C 180,E1 -10161.043,E2 -10161.043} C_VEL
LIN {X 0,Y 417.37,Z 841.716,A -85,B 0,C 180,E1 -10162.258,E2 -10162.258} C_VEL
LIN {X 0,Y 417.256,Z 846.245,A -85,B 0,C 180,E1 -10163.597,E2 -10163.597} C_VEL
LIN {X 0,Y 417.198,Z 850.36,A -85,B 0,C 180,E1 -10165.168,E2 -10165.168} C_VEL
LIN {X 0,Y 417.199,Z 852.299,A -85,B 0,C 180,E1 -10166.136,E2 -10166.136} C_VEL
LIN {X 0,Y 417.281,Z 853.767,A -85,B 0,C 180,E1 -10167.104,E2 -10167.104} C_VEL
LIN {X 0,Y 417.304,Z 854.818,A -85,B 0,C 180,E1 -10168.07,E2 -10168.07} C_VEL
LIN {X 0,Y 417.209,Z 855.459,A -85,B 0,C 180,E1 -10169.035,E2 -10169.035} C_VEL
LIN {X 0,Y 417.182,Z 855.687,A -85,B 0,C 180,E1 -10170,E2 -10170} C_VEL
LIN {X 0,Y 417.303,Z 854.872,A -85,B 0,C 180,E1 -10171.93,E2 -10171.93} C_VEL
LIN {X 0,Y 417.282,Z 853.855,A -85,B 0,C 180,E1 -10172.896,E2 -10172.896} C_VEL
LIN {X 0,Y 417.21,Z 852.396,A -85,B 0,C 180,E1 -10173.863,E2 -10173.863} C_VEL
LIN {X 0,Y 417.26,Z 849.38,A -85,B 0,C 180,E1 -10175.315,E2 -10175.315} C_VEL
LIN {X 0,Y 417.254,Z 845.273,A -85,B 0,C 180,E1 -10176.771,E2 -10176.771} C_VEL
LIN {X 0,Y 417.472,Z 838.952,A -85,B 0,C 180,E1 -10178.47,E2 -10178.47} C_VEL
LIN {X 0,Y 417.763,Z 832.063,A -85,B 0,C 180,E1 -10179.929,E2 -10179.929} C_VEL
LIN {X 0,Y 418.299,Z 823.495,A -85,B 0,C 180,E1 -10181.386,E2 -10181.386} C_VEL
LIN {X 0,Y 418.852,Z 814.668,A -85,B 0,C 180,E1 -10182.599,E2 -10182.599} C_VEL
LIN {X 0,Y 419.508,Z 803.807,A -85,B 0,C 180,E1 -10183.811,E2 -10183.811} C_VEL
LIN {X 0,Y 420.264,Z 792.982,A -85,B 0,C 180,E1 -10184.775,E2 -10184.775} C_VEL
LIN {X 0,Y 421.066,Z 780.942,A -85,B 0,C 180,E1 -10185.613,E2 -10185.613} C_VEL
LIN {X 0,Y 421.708,Z 768.37,A -85,B 0,C 180,E1 -10186.271,E2 -10186.271} C_VEL
LIN {X 0,Y 422.287,Z 755.155,A -85,B 0,C 180,E1 -10186.745,E2 -10186.745} C_VEL
LIN {X 0,Y 422.615,Z 740.092,A -85,B 0,C 180,E1 -10187.074,E2 -10187.074} C_VEL
LIN {X 0,Y 423.384,Z 668.694,A -85,B 0,C 180,E1 -10188.337,E2 -10188.337} C_VEL
LIN {X 0,Y 420.088,Z 640.914,A -85,B 0,C 180,E1 -10188.989,E2 -10188.989} C_VEL
LIN {X 0,Y 421.197,Z 621.82,A -85,B 0,C 180,E1 -10191.793,E2 -10191.793} C_VEL
LIN {X 0,Y 422.68,Z 599.627,A -85,B 0,C 180,E1 -10195.086,E2 -10195.086} C_VEL
LIN {X 0,Y 422.295,Z 596.149,A -85,B 0,C 180,E1 -10195.638,E2 -10195.638} C_VEL
LIN {X 0,Y 418.736,Z 580.223,A -85,B 0,C 180,E1 -10198.303,E2 -10198.303} C_VEL
LIN {X 0,Y 418.289,Z 578.381,A -85,B 0,C 180,E1 -10198.64,E2 -10198.64} C_VEL
LIN {X 0,Y 418.211,Z 578.392,A -85,B 0,C 180,E1 -10201.395,E2 -10201.395} C_VEL
LIN {X 0,Y 418.264,Z 578.383,A -85,B 0,C 180,E1 -10204.58,E2 -10204.58} C_VEL
LIN {X 0,Y 418.235,Z 578.387,A -85,B 0,C 180,E1 -10207.834,E2 -10207.834} C_VEL
LIN {X 0,Y 418.262,Z 578.38,A -85,B 0,C 180,E1 -10210.942,E2 -10210.942} C_VEL
LIN {X 0,Y 418.206,Z 578.391,A -85,B 0,C 180,E1 -10213.729,E2 -10213.729} C_VEL
LIN {X 0,Y 418.279,Z 578.38,A -85,B 0,C 180,E1 -10216.458,E2 -10216.458} C_VEL
LIN {X 0,Y 418.262,Z 578.379,A -85,B 0,C 180,E1 -10219.122,E2 -10219.122} C_VEL
LIN {X 0,Y 418.233,Z 578.388,A -85,B 0,C 180,E1 -10222.164,E2 -10222.164} C_VEL
LIN {X 0,Y 418.26,Z 578.372,A -85,B 0,C 180,E1 -10225.419,E2 -10225.419} C_VEL
LIN {X 0,Y 418.216,Z 578.389,A -85,B 0,C 180,E1 -10228.604,E2 -10228.604} C_VEL
LIN {X 0,Y 418.288,Z 578.37,A -85,B 0,C 180,E1 -10231.936,E2 -10231.936} C_VEL
LIN {X 0,Y 418.282,Z 578.377,A -85,B 0,C 180,E1 -10235.162,E2 -10235.162} C_VEL
LIN {X 0,Y 418.225,Z 578.379,A -85,B 0,C 180,E1 -10238.303,E2 -10238.303} C_VEL
LIN {X 0,Y 418.275,Z 578.379,A -85,B 0,C 180,E1 -10241.383,E2 -10241.383} C_VEL
LIN {X 0,Y 418.293,Z 578.369,A -85,B 0,C 180,E1 -10244.406,E2 -10244.406} C_VEL
LIN {X 0,Y 418.346,Z 578.37,A -85,B 0,C 180,E1 -10247.385,E2 -10247.385} C_VEL
LIN {X 0,Y 418.333,Z 578.367,A -85,B 0,C 180,E1 -10250.328,E2 -10250.328} C_VEL
LIN {X 0,Y 418.486,Z 578.353,A -85,B 0,C 180,E1 -10253.249,E2 -10253.249} C_VEL
LIN {X 0,Y 418.338,Z 578.372,A -85,B 0,C 180,E1 -10255.182,E2 -10255.182} C_VEL
LIN {X 0,Y 418.536,Z 578.338,A -85,B 0,C 180,E1 -10258.075,E2 -10258.075} C_VEL
LIN {X 0,Y 418.665,Z 578.325,A -85,B 0,C 180,E1 -10260,E2 -10260} C_VEL
LIN {X 0,Y 418.503,Z 578.354,A -85,B 0,C 180,E1 -10262.888,E2 -10262.888} C_VEL
LIN {X 0,Y 418.485,Z 578.347,A -85,B 0,C 180,E1 -10266.751,E2 -10266.751} C_VEL
LIN {X 0,Y 418.333,Z 578.372,A -85,B 0,C 180,E1 -10269.672,E2 -10269.672} C_VEL
LIN {X 0,Y 418.337,Z 578.366,A -85,B 0,C 180,E1 -10273.001,E2 -10273.001} C_VEL
LIN {X 0,Y 418.304,Z 578.381,A -85,B 0,C 180,E1 -10276.736,E2 -10276.736} C_VEL
LIN {X 0,Y 418.262,Z 578.376,A -85,B 0,C 180,E1 -10279.791,E2 -10279.791} C_VEL
LIN {X 0,Y 418.224,Z 578.39,A -85,B 0,C 180,E1 -10282.737,E2 -10282.737} C_VEL
LIN {X 0,Y 418.264,Z 578.379,A -85,B 0,C 180,E1 -10285.905,E2 -10285.905} C_VEL
LIN {X 0,Y 418.268,Z 578.378,A -85,B 0,C 180,E1 -10289.162,E2 -10289.162} C_VEL
LIN {X 0,Y 418.254,Z 578.387,A -85,B 0,C 180,E1 -10292.845,E2 -10292.845} C_VEL
LIN {X 0,Y 418.243,Z 578.384,A -85,B 0,C 180,E1 -10296.239,E2 -10296.239} C_VEL
LIN {X 0,Y 418.257,Z 578.381,A -85,B 0,C 180,E1 -10299.681,E2 -10299.681} C_VEL
LIN {X 0,Y 418.242,Z 578.365,A -85,B 0,C 180,E1 -10302.325,E2 -10302.325} C_VEL
LIN {X 0,Y 418.234,Z 578.389,A -85,B 0,C 180,E1 -10305.11,E2 -10305.11} C_VEL
LIN {X 0,Y 418.236,Z 578.375,A -85,B 0,C 180,E1 -10307.768,E2 -10307.768} C_VEL
LIN {X 0,Y 418.256,Z 578.377,A -85,B 0,C 180,E1 -10311.56,E2 -10311.56} C_VEL
LIN {X 0,Y 418.258,Z 578.386,A -85,B 0,C 180,E1 -10315.16,E2 -10315.16} C_VEL
LIN {X 0,Y 418.243,Z 578.385,A -85,B 0,C 180,E1 -10318.607,E2 -10318.607} C_VEL
LIN {X 0,Y 418.228,Z 578.387,A -85,B 0,C 180,E1 -10318.76,E2 -10318.76} C_VEL
LIN {X 0,Y 420.014,Z 583.083,A -85,B 0,C 180,E1 -10318.953,E2 -10318.953} C_VEL
LIN {X 0,Y 424.588,Z 594.021,A -85,B 0,C 180,E1 -10319.399,E2 -10319.399} C_VEL
LIN {X 0,Y 423.526,Z 679.941,A -85,B 0,C 180,E1 -10320.896,E2 -10320.896} C_VEL
LIN {X 0,Y 423.296,Z 692.312,A -85,B 0,C 180,E1 -10321.282,E2 -10321.282} C_VEL
LIN {X 0,Y 422.893,Z 704.91,A -85,B 0,C 180,E1 -10321.871,E2 -10321.871} C_VEL
LIN {X 0,Y 422.322,Z 716.815,A -85,B 0,C 180,E1 -10322.632,E2 -10322.632} C_VEL
LIN {X 0,Y 421.615,Z 727.68,A -85,B 0,C 180,E1 -10323.52,E2 -10323.52} C_VEL
LIN {X 0,Y 420.89,Z 737.347,A -85,B 0,C 180,E1 -10324.502,E2 -10324.502} C_VEL
LIN {X 0,Y 420.274,Z 745.791,A -85,B 0,C 180,E1 -10325.552,E2 -10325.552} C_VEL
LIN {X 0,Y 419.501,Z 755.142,A -85,B 0,C 180,E1 -10326.984,E2 -10326.984} C_VEL
LIN {X 0,Y 418.916,Z 762.304,A -85,B 0,C 180,E1 -10328.341,E2 -10328.341} C_VEL
LIN {X 0,Y 418.401,Z 768.729,A -85,B 0,C 180,E1 -10329.854,E2 -10329.854} C_VEL
LIN {X 0,Y 417.98,Z 773.752,A -85,B 0,C 180,E1 -10331.37,E2 -10331.37} C_VEL
LIN {X 0,Y 417.714,Z 777.552,A -85,B 0,C 180,E1 -10332.877,E2 -10332.877} C_VEL
LIN {X 0,Y 417.475,Z 780.274,A -85,B 0,C 180,E1 -10334.375,E2 -10334.375} C_VEL
LIN {X 0,Y 417.352,Z 781.534,A -85,B 0,C 180,E1 -10335.369,E2 -10335.369} C_VEL
LIN {X 0,Y 417.273,Z 782.389,A -85,B 0,C 180,E1 -10336.362,E2 -10336.362} C_VEL
LIN {X 0,Y 417.285,Z 782.826,A -85,B 0,C 180,E1 -10337.648,E2 -10337.648} C_VEL
LIN {X 0,Y 417.269,Z 782.405,A -85,B 0,C 180,E1 -10339.323,E2 -10339.323} C_VEL
LIN {X 0,Y 417.295,Z 781.603,A -85,B 0,C 180,E1 -10340.304,E2 -10340.304} C_VEL
LIN {X 0,Y 417.507,Z 778.75,A -85,B 0,C 180,E1 -10342.261,E2 -10342.261} C_VEL
LIN {X 0,Y 417.711,Z 775.291,A -85,B 0,C 180,E1 -10343.792,E2 -10343.792} C_VEL
LIN {X 0,Y 417.13,Z 773.266,A -85,B 0,C 180,E1 -10344.547,E2 -10344.547} C_VEL
LIN {X 0,Y 414.53,Z 769.545,A -85,B 0,C 180,E1 -10345.766,E2 -10345.766} C_VEL
LIN {X 0,Y 412.018,Z 765.239,A -85,B 0,C 180,E1 -10346.954,E2 -10346.954} C_VEL
LIN {X 0,Y 411.576,Z 762.141,A -85,B 0,C 180,E1 -10347.652,E2 -10347.652} C_VEL
LIN {X 0,Y 412.043,Z 754.846,A -85,B 0,C 180,E1 -10349.023,E2 -10349.023} C_VEL
LIN {X 0,Y 412.72,Z 746.884,A -85,B 0,C 180,E1 -10350.244,E2 -10350.244} C_VEL
LIN {X 0,Y 413.377,Z 737.221,A -85,B 0,C 180,E1 -10351.461,E2 -10351.461} C_VEL
LIN {X 0,Y 414.024,Z 726.37,A -85,B 0,C 180,E1 -10352.554,E2 -10352.554} C_VEL
LIN {X 0,Y 414.711,Z 715.776,A -85,B 0,C 180,E1 -10353.4,E2 -10353.4} C_VEL
LIN {X 0,Y 415.255,Z 703.069,A -85,B 0,C 180,E1 -10354.185,E2 -10354.185} C_VEL
LIN {X 0,Y 415.653,Z 690.073,A -85,B 0,C 180,E1 -10354.758,E2 -10354.758} C_VEL
LIN {X 0,Y 415.939,Z 677.386,A -85,B 0,C 180,E1 -10355.12,E2 -10355.12} C_VEL
LIN {X 0,Y 416.817,Z 594.692,A -85,B 0,C 180,E1 -10356.551,E2 -10356.551} C_VEL
LIN {X 0,Y 411.434,Z 579.235,A -85,B 0,C 180,E1 -10357.059,E2 -10357.059} C_VEL
LIN {X 0,Y 411.297,Z 579.253,A -85,B 0,C 180,E1 -10359.838,E2 -10359.838} C_VEL
LIN {X 0,Y 411.316,Z 579.246,A -85,B 0,C 180,E1 -10363.109,E2 -10363.109} C_VEL
LIN {X 0,Y 411.259,Z 579.255,A -85,B 0,C 180,E1 -10366.888,E2 -10366.888} C_VEL
LIN {X 0,Y 411.232,Z 579.263,A -85,B 0,C 180,E1 -10369.986,E2 -10369.986} C_VEL
LIN {X 0,Y 411.196,Z 579.261,A -85,B 0,C 180,E1 -10373.147,E2 -10373.147} C_VEL
LIN {X 0,Y 411.261,Z 579.255,A -85,B 0,C 180,E1 -10376.652,E2 -10376.652} C_VEL
LIN {X 0,Y 411.29,Z 579.252,A -85,B 0,C 180,E1 -10376.821,E2 -10376.821} C_VEL
LIN {X 0,Y 414.215,Z 587.423,A -85,B 0,C 180,E1 -10377.138,E2 -10377.138} C_VEL
LIN {X 0,Y 417.109,Z 595.085,A -85,B 0,C 180,E1 -10377.414,E2 -10377.414} C_VEL
LIN {X 0,Y 415.911,Z 681.034,A -85,B 0,C 180,E1 -10378.998,E2 -10378.998} C_VEL
LIN {X 0,Y 415.597,Z 694.444,A -85,B 0,C 180,E1 -10379.453,E2 -10379.453} C_VEL
LIN {X 0,Y 415.188,Z 706.666,A -85,B 0,C 180,E1 -10380.062,E2 -10380.062} C_VEL
LIN {X 0,Y 414.597,Z 718.401,A -85,B 0,C 180,E1 -10380.848,E2 -10380.848} C_VEL
LIN {X 0,Y 413.902,Z 730.535,A -85,B 0,C 180,E1 -10381.897,E2 -10381.897} C_VEL
LIN {X 0,Y 413.263,Z 740.389,A -85,B 0,C 180,E1 -10382.969,E2 -10382.969} C_VEL
LIN {X 0,Y 412.58,Z 749.591,A -85,B 0,C 180,E1 -10384.202,E2 -10384.202} C_VEL
LIN {X 0,Y 412.019,Z 757.223,A -85,B 0,C 180,E1 -10385.446,E2 -10385.446} C_VEL
LIN {X 0,Y 411.419,Z 765.075,A -85,B 0,C 180,E1 -10387.023,E2 -10387.023} C_VEL
LIN {X 0,Y 411.012,Z 771.461,A -85,B 0,C 180,E1 -10388.668,E2 -10388.668} C_VEL
LIN {X 0,Y 410.68,Z 775.741,A -85,B 0,C 180,E1 -10390.075,E2 -10390.075} C_VEL
LIN {X 0,Y 410.421,Z 779.804,A -85,B 0,C 180,E1 -10391.899,E2 -10391.899} C_VEL
LIN {X 0,Y 410.249,Z 781.867,A -85,B 0,C 180,E1 -10393.253,E2 -10393.253} C_VEL
LIN {X 0,Y 410.184,Z 783.174,A -85,B 0,C 180,E1 -10394.625,E2 -10394.625} C_VEL
LIN {X 0,Y 410.164,Z 783.691,A -85,B 0,C 180,E1 -10396.024,E2 -10396.024} C_VEL
LIN {X 0,Y 410.224,Z 782.966,A -85,B 0,C 180,E1 -10398.075,E2 -10398.075} C_VEL
LIN {X 0,Y 410.331,Z 781.6,A -85,B 0,C 180,E1 -10399.394,E2 -10399.394} C_VEL
LIN {X 0,Y 410.532,Z 779.512,A -85,B 0,C 180,E1 -10400.697,E2 -10400.697} C_VEL
LIN {X 0,Y 410.92,Z 774.975,A -85,B 0,C 180,E1 -10402.615,E2 -10402.615} C_VEL
LIN {X 0,Y 411.248,Z 770.649,A -85,B 0,C 180,E1 -10403.977,E2 -10403.977} C_VEL
LIN {X 0,Y 411.674,Z 765.034,A -85,B 0,C 180,E1 -10405.391,E2 -10405.391} C_VEL
LIN {X 0,Y 412.3,Z 757.315,A -85,B 0,C 180,E1 -10406.943,E2 -10406.943} C_VEL
LIN {X 0,Y 413.044,Z 748.916,A -85,B 0,C 180,E1 -10408.292,E2 -10408.292} C_VEL
LIN {X 0,Y 413.768,Z 739.345,A -85,B 0,C 180,E1 -10409.534,E2 -10409.534} C_VEL
LIN {X 0,Y 414.527,Z 728.159,A -85,B 0,C 180,E1 -10410.703,E2 -10410.703} C_VEL
LIN {X 0,Y 415.213,Z 716.37,A -85,B 0,C 180,E1 -10411.66,E2 -10411.66} C_VEL
LIN {X 0,Y 415.841,Z 703.736,A -85,B 0,C 180,E1 -10412.441,E2 -10412.441} C_VEL
LIN {X 0,Y 416.182,Z 691.073,A -85,B 0,C 180,E1 -10413.009,E2 -10413.009} C_VEL
LIN {X 0,Y 416.451,Z 678.268,A -85,B 0,C 180,E1 -10413.377,E2 -10413.377} C_VEL
LIN {X 0,Y 417.616,Z 595.233,A -85,B 0,C 180,E1 -10414.92,E2 -10414.92} C_VEL
LIN {X 0,Y 411.328,Z 579.771,A -85,B 0,C 180,E1 -10415.57,E2 -10415.57} C_VEL
LIN {X 0,Y 411.266,Z 579.257,A -85,B 0,C 180,E1 -10415.598,E2 -10415.598} C_VEL
LIN {X 0,Y 411.188,Z 579.268,A -85,B 0,C 180,E1 -10418.965,E2 -10418.965} C_VEL
LIN {X 0,Y 411.244,Z 579.26,A -85,B 0,C 180,E1 -10422.084,E2 -10422.084} C_VEL
LIN {X 0,Y 411.254,Z 579.258,A -85,B 0,C 180,E1 -10425.147,E2 -10425.147} C_VEL
LIN {X 0,Y 411.293,Z 579.254,A -85,B 0,C 180,E1 -10428.167,E2 -10428.167} C_VEL
LIN {X 0,Y 411.473,Z 579.231,A -85,B 0,C 180,E1 -10432.146,E2 -10432.146} C_VEL
LIN {X 0,Y 411.483,Z 579.23,A -85,B 0,C 180,E1 -10434.118,E2 -10434.118} C_VEL
LIN {X 0,Y 411.505,Z 579.223,A -85,B 0,C 180,E1 -10438.043,E2 -10438.043} C_VEL
LIN {X 0,Y 411.634,Z 579.209,A -85,B 0,C 180,E1 -10440,E2 -10440} C_VEL
LIN {X 0,Y 411.458,Z 579.228,A -85,B 0,C 180,E1 -10442.937,E2 -10442.937} C_VEL
LIN {X 0,Y 411.484,Z 579.227,A -85,B 0,C 180,E1 -10445.882,E2 -10445.882} C_VEL
LIN {X 0,Y 411.348,Z 579.242,A -85,B 0,C 180,E1 -10448.845,E2 -10448.845} C_VEL
LIN {X 0,Y 411.29,Z 579.247,A -85,B 0,C 180,E1 -10451.833,E2 -10451.833} C_VEL
LIN {X 0,Y 411.254,Z 579.254,A -85,B 0,C 180,E1 -10454.853,E2 -10454.853} C_VEL
LIN {X 0,Y 411.244,Z 579.251,A -85,B 0,C 180,E1 -10457.915,E2 -10457.915} C_VEL
LIN {X 0,Y 411.19,Z 579.262,A -85,B 0,C 180,E1 -10461.035,E2 -10461.035} C_VEL
LIN {X 0,Y 411.219,Z 579.257,A -85,B 0,C 180,E1 -10464.216,E2 -10464.216} C_VEL
LIN {X 0,Y 411.253,Z 579.25,A -85,B 0,C 180,E1 -10467.478,E2 -10467.478} C_VEL
LIN {X 0,Y 411.191,Z 579.263,A -85,B 0,C 180,E1 -10470.848,E2 -10470.848} C_VEL
LIN {X 0,Y 411.2,Z 579.262,A -85,B 0,C 180,E1 -10474.334,E2 -10474.334} C_VEL
LIN {X 0,Y 411.2,Z 579.263,A -85,B 0,C 180,E1 -10477.973,E2 -10477.973} C_VEL
LIN {X 0,Y 411.205,Z 579.26,A -85,B 0,C 180,E1 -10481.237,E2 -10481.237} C_VEL
LIN {X 0,Y 411.22,Z 579.264,A -85,B 0,C 180,E1 -10484.485,E2 -10484.485} C_VEL
LIN {X 0,Y 411.195,Z 579.266,A -85,B 0,C 180,E1 -10488.198,E2 -10488.198} C_VEL
LIN {X 0,Y 411.228,Z 579.262,A -85,B 0,C 180,E1 -10490.778,E2 -10490.778} C_VEL
LIN {X 0,Y 411.197,Z 579.267,A -85,B 0,C 180,E1 -10494.472,E2 -10494.472} C_VEL
LIN {X 0,Y 411.206,Z 579.264,A -85,B 0,C 180,E1 -10496.874,E2 -10496.874} C_VEL
LIN {X 0,Y 411.23,Z 579.395,A -85,B 0,C 180,E1 -10499.477,E2 -10499.477} C_VEL
LIN {X 0,Y 413.973,Z 591.633,A -85,B 0,C 180,E1 -10501.983,E2 -10501.983} C_VEL
LIN {X 0,Y 415.301,Z 598.929,A -85,B 0,C 180,E1 -10503.411,E2 -10503.411} C_VEL
LIN {X 0,Y 414.305,Z 613.424,A -85,B 0,C 180,E1 -10505.977,E2 -10505.977} C_VEL
LIN {X 0,Y 413.022,Z 633.624,A -85,B 0,C 180,E1 -10509.497,E2 -10509.497} C_VEL
LIN {X 0,Y 412.691,Z 639.293,A -85,B 0,C 180,E1 -10510.444,E2 -10510.444} C_VEL
LIN {X 0,Y 416.606,Z 668.911,A -85,B 0,C 180,E1 -10511.214,E2 -10511.214} C_VEL
LIN {X 0,Y 416.956,Z 674.913,A -85,B 0,C 180,E1 -10511.346,E2 -10511.346} C_VEL
LIN {X 0,Y 415.88,Z 749.642,A -85,B 0,C 180,E1 -10512.736,E2 -10512.736} C_VEL
LIN {X 0,Y 415.3,Z 763.352,A -85,B 0,C 180,E1 -10513.186,E2 -10513.186} C_VEL
LIN {X 0,Y 414.436,Z 776.331,A -85,B 0,C 180,E1 -10513.815,E2 -10513.815} C_VEL
LIN {X 0,Y 413.742,Z 788.217,A -85,B 0,C 180,E1 -10514.609,E2 -10514.609} C_VEL
LIN {X 0,Y 412.901,Z 799.716,A -85,B 0,C 180,E1 -10515.586,E2 -10515.586} C_VEL
LIN {X 0,Y 412.276,Z 810.523,A -85,B 0,C 180,E1 -10516.742,E2 -10516.742} C_VEL
LIN {X 0,Y 411.506,Z 819.526,A -85,B 0,C 180,E1 -10517.924,E2 -10517.924} C_VEL
LIN {X 0,Y 410.858,Z 828.694,A -85,B 0,C 180,E1 -10519.404,E2 -10519.404} C_VEL
LIN {X 0,Y 410.472,Z 836.103,A -85,B 0,C 180,E1 -10520.888,E2 -10520.888} C_VEL
LIN {X 0,Y 410.297,Z 841.119,A -85,B 0,C 180,E1 -10522.124,E2 -10522.124} C_VEL
LIN {X 0,Y 410.168,Z 846.042,A -85,B 0,C 180,E1 -10523.617,E2 -10523.617} C_VEL
LIN {X 0,Y 410.136,Z 849.759,A -85,B 0,C 180,E1 -10525.085,E2 -10525.085} C_VEL
LIN {X 0,Y 410.11,Z 851.691,A -85,B 0,C 180,E1 -10526.07,E2 -10526.07} C_VEL
LIN {X 0,Y 410.208,Z 853.156,A -85,B 0,C 180,E1 -10527.054,E2 -10527.054} C_VEL
LIN {X 0,Y 410.251,Z 854.208,A -85,B 0,C 180,E1 -10528.037,E2 -10528.037} C_VEL
LIN {X 0,Y 410.155,Z 854.847,A -85,B 0,C 180,E1 -10529.018,E2 -10529.018} C_VEL
LIN {X 0,Y 410.126,Z 855.067,A -85,B 0,C 180,E1 -10530,E2 -10530} C_VEL
LIN {X 0,Y 410.251,Z 854.246,A -85,B 0,C 180,E1 -10531.963,E2 -10531.963} C_VEL
LIN {X 0,Y 410.21,Z 853.224,A -85,B 0,C 180,E1 -10532.946,E2 -10532.946} C_VEL
LIN {X 0,Y 410.121,Z 851.752,A -85,B 0,C 180,E1 -10533.93,E2 -10533.93} C_VEL
LIN {X 0,Y 410.168,Z 848.722,A -85,B 0,C 180,E1 -10535.407,E2 -10535.407} C_VEL
LIN {X 0,Y 410.176,Z 844.598,A -85,B 0,C 180,E1 -10536.888,E2 -10536.888} C_VEL
LIN {X 0,Y 410.4,Z 838.252,A -85,B 0,C 180,E1 -10538.618,E2 -10538.618} C_VEL
LIN {X 0,Y 410.717,Z 831.337,A -85,B 0,C 180,E1 -10540.101,E2 -10540.101} C_VEL
LIN {X 0,Y 411.297,Z 822.732,A -85,B 0,C 180,E1 -10541.582,E2 -10541.582} C_VEL
LIN {X 0,Y 411.906,Z 813.884,A -85,B 0,C 180,E1 -10542.815,E2 -10542.815} C_VEL
LIN {X 0,Y 412.559,Z 802.946,A -85,B 0,C 180,E1 -10544.049,E2 -10544.049} C_VEL
LIN {X 0,Y 413.329,Z 792.037,A -85,B 0,C 180,E1 -10545.028,E2 -10545.028} C_VEL
LIN {X 0,Y 414.219,Z 780.41,A -85,B 0,C 180,E1 -10545.878,E2 -10545.878} C_VEL
LIN {X 0,Y 414.901,Z 768.313,A -85,B 0,C 180,E1 -10546.546,E2 -10546.546} C_VEL
LIN {X 0,Y 415.524,Z 755.955,A -85,B 0,C 180,E1 -10547.026,E2 -10547.026} C_VEL
LIN {X 0,Y 415.893,Z 741.828,A -85,B 0,C 180,E1 -10547.359,E2 -10547.359} C_VEL
LIN {X 0,Y 416.566,Z 668.714,A -85,B 0,C 180,E1 -10548.652,E2 -10548.652} C_VEL
LIN {X 0,Y 413.2,Z 639.741,A -85,B 0,C 180,E1 -10549.389,E2 -10549.389} C_VEL
LIN {X 0,Y 414.444,Z 619.421,A -85,B 0,C 180,E1 -10552.429,E2 -10552.429} C_VEL
LIN {X 0,Y 415.791,Z 600.645,A -85,B 0,C 180,E1 -10555.264,E2 -10555.264} C_VEL
LIN {X 0,Y 414.58,Z 593.624,A -85,B 0,C 180,E1 -10556.422,E2 -10556.422} C_VEL
LIN {X 0,Y 411.256,Z 579.258,A -85,B 0,C 180,E1 -10558.919,E2 -10558.919} C_VEL
LIN {X 0,Y 411.164,Z 579.271,A -85,B 0,C 180,E1 -10561.996,E2 -10561.996} C_VEL
LIN {X 0,Y 411.21,Z 579.261,A -85,B 0,C 180,E1 -10564.878,E2 -10564.878} C_VEL
LIN {X 0,Y 411.212,Z 579.26,A -85,B 0,C 180,E1 -10568.169,E2 -10568.169} C_VEL
LIN {X 0,Y 411.197,Z 579.26,A -85,B 0,C 180,E1 -10571.233,E2 -10571.233} C_VEL
LIN {X 0,Y 411.181,Z 579.264,A -85,B 0,C 180,E1 -10574.488,E2 -10574.488} C_VEL
LIN {X 0,Y 411.228,Z 579.257,A -85,B 0,C 180,E1 -10577.296,E2 -10577.296} C_VEL
LIN {X 0,Y 411.227,Z 579.255,A -85,B 0,C 180,E1 -10580.777,E2 -10580.777} C_VEL
LIN {X 0,Y 411.194,Z 579.257,A -85,B 0,C 180,E1 -10584.471,E2 -10584.471} C_VEL
LIN {X 0,Y 411.165,Z 579.268,A -85,B 0,C 180,E1 -10588.003,E2 -10588.003} C_VEL
LIN {X 0,Y 411.217,Z 579.248,A -85,B 0,C 180,E1 -10591.41,E2 -10591.41} C_VEL
LIN {X 0,Y 411.229,Z 579.259,A -85,B 0,C 180,E1 -10594.706,E2 -10594.706} C_VEL
LIN {X 0,Y 411.197,Z 579.25,A -85,B 0,C 180,E1 -10597.913,E2 -10597.913} C_VEL
LIN {X 0,Y 411.216,Z 579.259,A -85,B 0,C 180,E1 -10601.051,E2 -10601.051} C_VEL
LIN {X 0,Y 411.245,Z 579.245,A -85,B 0,C 180,E1 -10604.131,E2 -10604.131} C_VEL
LIN {X 0,Y 411.294,Z 579.25,A -85,B 0,C 180,E1 -10607.165,E2 -10607.165} C_VEL
LIN {X 0,Y 411.285,Z 579.246,A -85,B 0,C 180,E1 -10610.161,E2 -10610.161} C_VEL
LIN {X 0,Y 411.449,Z 579.23,A -85,B 0,C 180,E1 -10613.133,E2 -10613.133} C_VEL
LIN {X 0,Y 411.31,Z 579.248,A -85,B 0,C 180,E1 -10615.099,E2 -10615.099} C_VEL
LIN {X 0,Y 411.505,Z 579.213,A -85,B 0,C 180,E1 -10618.043,E2 -10618.043} C_VEL
LIN {X 0,Y 411.634,Z 579.2,A -85,B 0,C 180,E1 -10620,E2 -10620} C_VEL
LIN {X 0,Y 411.458,Z 579.231,A -85,B 0,C 180,E1 -10622.937,E2 -10622.937} C_VEL
LIN {X 0,Y 411.442,Z 579.222,A -85,B 0,C 180,E1 -10626.625,E2 -10626.625} C_VEL
LIN {X 0,Y 411.285,Z 579.25,A -85,B 0,C 180,E1 -10629.839,E2 -10629.839} C_VEL
LIN {X 0,Y 411.296,Z 579.243,A -85,B 0,C 180,E1 -10633.104,E2 -10633.104} C_VEL
LIN {X 0,Y 411.254,Z 579.257,A -85,B 0,C 180,E1 -10636.869,E2 -10636.869} C_VEL
LIN {X 0,Y 411.222,Z 579.253,A -85,B 0,C 180,E1 -10639.987,E2 -10639.987} C_VEL
LIN {X 0,Y 411.189,Z 579.262,A -85,B 0,C 180,E1 -10643.148,E2 -10643.148} C_VEL
LIN {X 0,Y 411.231,Z 579.256,A -85,B 0,C 180,E1 -10646.381,E2 -10646.381} C_VEL
LIN {X 0,Y 411.205,Z 579.254,A -85,B 0,C 180,E1 -10649.712,E2 -10649.712} C_VEL
LIN {X 0,Y 411.201,Z 579.263,A -85,B 0,C 180,E1 -10653.156,E2 -10653.156} C_VEL
LIN {X 0,Y 411.19,Z 579.264,A -85,B 0,C 180,E1 -10656.554,E2 -10656.554} C_VEL
LIN {X 0,Y 411.219,Z 579.257,A -85,B 0,C 180,E1 -10659.731,E2 -10659.731} C_VEL
LIN {X 0,Y 411.177,Z 579.25,A -85,B 0,C 180,E1 -10663.133,E2 -10663.133} C_VEL
LIN {X 0,Y 411.164,Z 579.265,A -85,B 0,C 180,E1 -10665.882,E2 -10665.882} C_VEL
LIN {X 0,Y 411.16,Z 579.26,A -85,B 0,C 180,E1 -10668.773,E2 -10668.773} C_VEL
LIN {X 0,Y 411.197,Z 579.255,A -85,B 0,C 180,E1 -10672.028,E2 -10672.028} C_VEL
LIN {X 0,Y 411.204,Z 579.264,A -85,B 0,C 180,E1 -10675.667,E2 -10675.667} C_VEL
LIN {X 0,Y 411.189,Z 579.286,A -85,B 0,C 180,E1 -10678.382,E2 -10678.382} C_VEL
LIN {X 0,Y 413.015,Z 584.095,A -85,B 0,C 180,E1 -10678.577,E2 -10678.577} C_VEL
LIN {X 0,Y 418.047,Z 595.9,A -85,B 0,C 180,E1 -10679.077,E2 -10679.077} C_VEL
LIN {X 0,Y 416.873,Z 680.111,A -85,B 0,C 180,E1 -10680.562,E2 -10680.562} C_VEL
LIN {X 0,Y 416.619,Z 692.651,A -85,B 0,C 180,E1 -10680.955,E2 -10680.955} C_VEL
LIN {X 0,Y 416.229,Z 705.145,A -85,B 0,C 180,E1 -10681.544,E2 -10681.544} C_VEL
LIN {X 0,Y 415.638,Z 716.787,A -85,B 0,C 180,E1 -10682.291,E2 -10682.291} C_VEL
LIN {X 0,Y 414.864,Z 727.759,A -85,B 0,C 180,E1 -10683.19,E2 -10683.19} C_VEL
LIN {X 0,Y 414.005,Z 738.81,A -85,B 0,C 180,E1 -10684.339,E2 -10684.339} C_VEL
LIN {X 0,Y 413.229,Z 748.75,A -85,B 0,C 180,E1 -10685.643,E2 -10685.643} C_VEL
LIN {X 0,Y 412.471,Z 757.507,A -85,B 0,C 180,E1 -10687.069,E2 -10687.069} C_VEL
LIN {X 0,Y 411.866,Z 764.447,A -85,B 0,C 180,E1 -10688.478,E2 -10688.478} C_VEL
LIN {X 0,Y 411.322,Z 770.54,A -85,B 0,C 180,E1 -10690.018,E2 -10690.018} C_VEL
LIN {X 0,Y 410.916,Z 775.289,A -85,B 0,C 180,E1 -10691.555,E2 -10691.555} C_VEL
LIN {X 0,Y 410.648,Z 778.85,A -85,B 0,C 180,E1 -10693.086,E2 -10693.086} C_VEL
LIN {X 0,Y 410.485,Z 780.636,A -85,B 0,C 180,E1 -10694.102,E2 -10694.102} C_VEL
LIN {X 0,Y 410.308,Z 781.953,A -85,B 0,C 180,E1 -10695.112,E2 -10695.112} C_VEL
LIN {X 0,Y 410.234,Z 782.864,A -85,B 0,C 180,E1 -10696.123,E2 -10696.123} C_VEL
LIN {X 0,Y 410.228,Z 783.423,A -85,B 0,C 180,E1 -10697.56,E2 -10697.56} C_VEL
LIN {X 0,Y 410.214,Z 783.09,A -85,B 0,C 180,E1 -10699.137,E2 -10699.137} C_VEL
LIN {X 0,Y 410.231,Z 782.377,A -85,B 0,C 180,E1 -10700.136,E2 -10700.136} C_VEL
LIN {X 0,Y 410.291,Z 781.223,A -85,B 0,C 180,E1 -10701.132,E2 -10701.132} C_VEL
LIN {X 0,Y 410.602,Z 777.718,A -85,B 0,C 180,E1 -10703.096,E2 -10703.096} C_VEL
LIN {X 0,Y 410.794,Z 773.839,A -85,B 0,C 180,E1 -10704.601,E2 -10704.601} C_VEL
LIN {X 0,Y 411.057,Z 768.89,A -85,B 0,C 180,E1 -10706.079,E2 -10706.079} C_VEL
LIN {X 0,Y 411.576,Z 762.141,A -85,B 0,C 180,E1 -10707.652,E2 -10707.652} C_VEL
LIN {X 0,Y 411.16,Z 758.848,A -85,B 0,C 180,E1 -10708.332,E2 -10708.332} C_VEL
LIN {X 0,Y 408.804,Z 753.197,A -85,B 0,C 180,E1 -10709.425,E2 -10709.425} C_VEL
LIN {X 0,Y 406.484,Z 747.001,A -85,B 0,C 180,E1 -10710.463,E2 -10710.463} C_VEL
LIN {X 0,Y 406.118,Z 742.795,A -85,B 0,C 180,E1 -10711.045,E2 -10711.045} C_VEL
LIN {X 0,Y 406.776,Z 732.495,A -85,B 0,C 180,E1 -10712.228,E2 -10712.228} C_VEL
LIN {X 0,Y 407.486,Z 721.711,A -85,B 0,C 180,E1 -10713.213,E2 -10713.213} C_VEL
LIN {X 0,Y 408.165,Z 709.693,A -85,B 0,C 180,E1 -10714.073,E2 -10714.073} C_VEL
LIN {X 0,Y 408.657,Z 696.906,A -85,B 0,C 180,E1 -10714.747,E2 -10714.747} C_VEL
LIN {X 0,Y 408.955,Z 684.402,A -85,B 0,C 180,E1 -10715.207,E2 -10715.207} C_VEL
LIN {X 0,Y 409.155,Z 668.374,A -85,B 0,C 180,E1 -10715.544,E2 -10715.544} C_VEL
LIN {X 0,Y 409.934,Z 595.923,A -85,B 0,C 180,E1 -10716.814,E2 -10716.814} C_VEL
LIN {X 0,Y 404.386,Z 580.114,A -85,B 0,C 180,E1 -10717.346,E2 -10717.346} C_VEL
LIN {X 0,Y 404.264,Z 580.125,A -85,B 0,C 180,E1 -10721.024,E2 -10721.024} C_VEL
LIN {X 0,Y 404.219,Z 580.137,A -85,B 0,C 180,E1 -10724.088,E2 -10724.088} C_VEL
LIN {X 0,Y 404.205,Z 580.133,A -85,B 0,C 180,E1 -10727.192,E2 -10727.192} C_VEL
LIN {X 0,Y 404.165,Z 580.139,A -85,B 0,C 180,E1 -10730.351,E2 -10730.351} C_VEL
LIN {X 0,Y 404.163,Z 580.139,A -85,B 0,C 180,E1 -10733.574,E2 -10733.574} C_VEL
LIN {X 0,Y 404.207,Z 580.134,A -85,B 0,C 180,E1 -10736.527,E2 -10736.527} C_VEL
LIN {X 0,Y 410.412,Z 597.163,A -85,B 0,C 180,E1 -10737.151,E2 -10737.151} C_VEL
LIN {X 0,Y 409.103,Z 681.238,A -85,B 0,C 180,E1 -10738.723,E2 -10738.723} C_VEL
LIN {X 0,Y 408.781,Z 695.042,A -85,B 0,C 180,E1 -10739.197,E2 -10739.197} C_VEL
LIN {X 0,Y 408.384,Z 706.902,A -85,B 0,C 180,E1 -10739.795,E2 -10739.795} C_VEL
LIN {X 0,Y 407.775,Z 718.511,A -85,B 0,C 180,E1 -10740.577,E2 -10740.577} C_VEL
LIN {X 0,Y 407.051,Z 730.606,A -85,B 0,C 180,E1 -10741.63,E2 -10741.63} C_VEL
LIN {X 0,Y 406.361,Z 740.548,A -85,B 0,C 180,E1 -10742.714,E2 -10742.714} C_VEL
LIN {X 0,Y 405.65,Z 749.926,A -85,B 0,C 180,E1 -10743.982,E2 -10743.982} C_VEL
LIN {X 0,Y 405.02,Z 758.207,A -85,B 0,C 180,E1 -10745.357,E2 -10745.357} C_VEL
LIN {X 0,Y 404.396,Z 765.831,A -85,B 0,C 180,E1 -10746.924,E2 -10746.924} C_VEL
LIN {X 0,Y 404.012,Z 771.806,A -85,B 0,C 180,E1 -10748.482,E2 -10748.482} C_VEL
LIN {X 0,Y 403.627,Z 776.637,A -85,B 0,C 180,E1 -10750.108,E2 -10750.108} C_VEL
LIN {X 0,Y 403.413,Z 779.758,A -85,B 0,C 180,E1 -10751.486,E2 -10751.486} C_VEL
LIN {X 0,Y 403.213,Z 782.146,A -85,B 0,C 180,E1 -10752.94,E2 -10752.94} C_VEL
LIN {X 0,Y 403.125,Z 783.616,A -85,B 0,C 180,E1 -10754.374,E2 -10754.374} C_VEL
LIN {X 0,Y 403.101,Z 784.256,A -85,B 0,C 180,E1 -10755.782,E2 -10755.782} C_VEL
LIN {X 0,Y 403.134,Z 784.133,A -85,B 0,C 180,E1 -10757.164,E2 -10757.164} C_VEL
LIN {X 0,Y 403.203,Z 783.266,A -85,B 0,C 180,E1 -10758.546,E2 -10758.546} C_VEL
LIN {X 0,Y 403.391,Z 781.421,A -85,B 0,C 180,E1 -10760.046,E2 -10760.046} C_VEL
LIN {X 0,Y 403.654,Z 778.546,A -85,B 0,C 180,E1 -10761.58,E2 -10761.58} C_VEL
LIN {X 0,Y 403.993,Z 774.488,A -85,B 0,C 180,E1 -10763.15,E2 -10763.15} C_VEL
LIN {X 0,Y 404.496,Z 768.007,A -85,B 0,C 180,E1 -10765.015,E2 -10765.015} C_VEL
LIN {X 0,Y 405.058,Z 761.903,A -85,B 0,C 180,E1 -10766.388,E2 -10766.388} C_VEL
LIN {X 0,Y 405.763,Z 754.058,A -85,B 0,C 180,E1 -10767.824,E2 -10767.824} C_VEL
LIN {X 0,Y 406.513,Z 745.07,A -85,B 0,C 180,E1 -10769.147,E2 -10769.147} C_VEL
LIN {X 0,Y 407.338,Z 734.459,A -85,B 0,C 180,E1 -10770.404,E2 -10770.404} C_VEL
LIN {X 0,Y 408.108,Z 723.576,A -85,B 0,C 180,E1 -10771.431,E2 -10771.431} C_VEL
LIN {X 0,Y 408.762,Z 711.147,A -85,B 0,C 180,E1 -10772.34,E2 -10772.34} C_VEL
LIN {X 0,Y 409.275,Z 699.596,A -85,B 0,C 180,E1 -10772.977,E2 -10772.977} C_VEL
LIN {X 0,Y 409.569,Z 687.042,A -85,B 0,C 180,E1 -10773.476,E2 -10773.476} C_VEL
LIN {X 0,Y 409.839,Z 671.904,A -85,B 0,C 180,E1 -10773.826,E2 -10773.826} C_VEL
LIN {X 0,Y 410.98,Z 596.925,A -85,B 0,C 180,E1 -10775.245,E2 -10775.245} C_VEL
LIN {X 0,Y 404.277,Z 580.721,A -85,B 0,C 180,E1 -10775.956,E2 -10775.956} C_VEL
LIN {X 0,Y 404.184,Z 580.141,A -85,B 0,C 180,E1 -10776.018,E2 -10776.018} C_VEL
LIN {X 0,Y 404.183,Z 580.139,A -85,B 0,C 180,E1 -10779.874,E2 -10779.874} C_VEL
LIN {X 0,Y 404.207,Z 580.136,A -85,B 0,C 180,E1 -10782.993,E2 -10782.993} C_VEL
LIN {X 0,Y 404.274,Z 580.129,A -85,B 0,C 180,E1 -10786.939,E2 -10786.939} C_VEL
LIN {X 0,Y 404.263,Z 580.128,A -85,B 0,C 180,E1 -10789.988,E2 -10789.988} C_VEL
LIN {X 0,Y 404.404,Z 580.111,A -85,B 0,C 180,E1 -10793.013,E2 -10793.013} C_VEL
LIN {X 0,Y 404.281,Z 580.125,A -85,B 0,C 180,E1 -10795.014,E2 -10795.014} C_VEL
LIN {X 0,Y 404.474,Z 580.098,A -85,B 0,C 180,E1 -10798.008,E2 -10798.008} C_VEL
LIN {X 0,Y 404.604,Z 580.085,A -85,B 0,C 180,E1 -10800,E2 -10800} C_VEL
LIN {X 0,Y 404.416,Z 580.105,A -85,B 0,C 180,E1 -10802.988,E2 -10802.988} C_VEL
LIN {X 0,Y 404.43,Z 580.106,A -85,B 0,C 180,E1 -10805.985,E2 -10805.985} C_VEL
LIN {X 0,Y 404.287,Z 580.12,A -85,B 0,C 180,E1 -10809.001,E2 -10809.001} C_VEL
LIN {X 0,Y 404.261,Z 580.124,A -85,B 0,C 180,E1 -10812.041,E2 -10812.041} C_VEL
LIN {X 0,Y 404.199,Z 580.131,A -85,B 0,C 180,E1 -10815.118,E2 -10815.118} C_VEL
LIN {X 0,Y 404.202,Z 580.13,A -85,B 0,C 180,E1 -10818.239,E2 -10818.239} C_VEL
LIN {X 0,Y 404.132,Z 580.139,A -85,B 0,C 180,E1 -10821.42,E2 -10821.42} C_VEL
LIN {X 0,Y 404.17,Z 580.138,A -85,B 0,C 180,E1 -10824.666,E2 -10824.666} C_VEL
LIN {X 0,Y 404.191,Z 580.132,A -85,B 0,C 180,E1 -10828,E2 -10828} C_VEL
LIN {X 0,Y 404.136,Z 580.141,A -85,B 0,C 180,E1 -10831.56,E2 -10831.56} C_VEL
LIN {X 0,Y 404.18,Z 580.138,A -85,B 0,C 180,E1 -10835.017,E2 -10835.017} C_VEL
LIN {X 0,Y 404.159,Z 580.14,A -85,B 0,C 180,E1 -10838.757,E2 -10838.757} C_VEL
LIN {X 0,Y 404.187,Z 580.134,A -85,B 0,C 180,E1 -10841.612,E2 -10841.612} C_VEL
LIN {X 0,Y 404.185,Z 580.141,A -85,B 0,C 180,E1 -10844.529,E2 -10844.529} C_VEL
LIN {X 0,Y 404.167,Z 580.14,A -85,B 0,C 180,E1 -10847.301,E2 -10847.301} C_VEL
LIN {X 0,Y 404.166,Z 580.14,A -85,B 0,C 180,E1 -10849.956,E2 -10849.956} C_VEL
LIN {X 0,Y 404.138,Z 580.144,A -85,B 0,C 180,E1 -10853.125,E2 -10853.125} C_VEL
LIN {X 0,Y 404.143,Z 580.147,A -85,B 0,C 180,E1 -10856.189,E2 -10856.189} C_VEL
LIN {X 0,Y 404.153,Z 580.175,A -85,B 0,C 180,E1 -10859.101,E2 -10859.101} C_VEL
LIN {X 0,Y 406.981,Z 592.656,A -85,B 0,C 180,E1 -10861.727,E2 -10861.727} C_VEL
LIN {X 0,Y 408.335,Z 599.706,A -85,B 0,C 180,E1 -10863.142,E2 -10863.142} C_VEL
LIN {X 0,Y 408.015,Z 607.06,A -85,B 0,C 180,E1 -10864.494,E2 -10864.494} C_VEL
LIN {X 0,Y 406.336,Z 629.198,A -85,B 0,C 180,E1 -10868.437,E2 -10868.437} C_VEL
LIN {X 0,Y 405.796,Z 638.329,A -85,B 0,C 180,E1 -10870.048,E2 -10870.048} C_VEL
LIN {X 0,Y 409.872,Z 668.897,A -85,B 0,C 180,E1 -10870.881,E2 -10870.881} C_VEL
LIN {X 0,Y 410.252,Z 675.535,A -85,B 0,C 180,E1 -10871.03,E2 -10871.03} C_VEL
LIN {X 0,Y 409.122,Z 749.628,A -85,B 0,C 180,E1 -10872.441,E2 -10872.441} C_VEL
LIN {X 0,Y 408.507,Z 763.114,A -85,B 0,C 180,E1 -10872.898,E2 -10872.898} C_VEL
LIN {X 0,Y 407.631,Z 775.946,A -85,B 0,C 180,E1 -10873.537,E2 -10873.537} C_VEL
LIN {X 0,Y 406.892,Z 787.775,A -85,B 0,C 180,E1 -10874.343,E2 -10874.343} C_VEL
LIN {X 0,Y 405.991,Z 799.227,A -85,B 0,C 180,E1 -10875.335,E2 -10875.335} C_VEL
LIN {X 0,Y 405.371,Z 809.232,A -85,B 0,C 180,E1 -10876.418,E2 -10876.418} C_VEL
LIN {X 0,Y 404.504,Z 818.958,A -85,B 0,C 180,E1 -10877.712,E2 -10877.712} C_VEL
LIN {X 0,Y 403.842,Z 828.107,A -85,B 0,C 180,E1 -10879.218,E2 -10879.218} C_VEL
LIN {X 0,Y 403.429,Z 835.508,A -85,B 0,C 180,E1 -10880.727,E2 -10880.727} C_VEL
LIN {X 0,Y 403.223,Z 840.521,A -85,B 0,C 180,E1 -10881.985,E2 -10881.985} C_VEL
LIN {X 0,Y 403.072,Z 845.857,A -85,B 0,C 180,E1 -10883.648,E2 -10883.648} C_VEL
LIN {X 0,Y 403.073,Z 849.159,A -85,B 0,C 180,E1 -10884.999,E2 -10884.999} C_VEL
LIN {X 0,Y 403.023,Z 851.083,A -85,B 0,C 180,E1 -10886,E2 -10886} C_VEL
LIN {X 0,Y 403.137,Z 852.547,A -85,B 0,C 180,E1 -10887.002,E2 -10887.002} C_VEL
LIN {X 0,Y 403.182,Z 853.598,A -85,B 0,C 180,E1 -10888.002,E2 -10888.002} C_VEL
LIN {X 0,Y 403.103,Z 854.237,A -85,B 0,C 180,E1 -10889.001,E2 -10889.001} C_VEL
LIN {X 0,Y 403.072,Z 854.447,A -85,B 0,C 180,E1 -10890,E2 -10890} C_VEL
LIN {X 0,Y 403.199,Z 853.617,A -85,B 0,C 180,E1 -10891.998,E2 -10891.998} C_VEL
LIN {X 0,Y 403.139,Z 852.588,A -85,B 0,C 180,E1 -10892.998,E2 -10892.998} C_VEL
LIN {X 0,Y 403.035,Z 851.1,A -85,B 0,C 180,E1 -10894,E2 -10894} C_VEL
LIN {X 0,Y 403.081,Z 848.056,A -85,B 0,C 180,E1 -10895.503,E2 -10895.503} C_VEL
LIN {X 0,Y 403.083,Z 843.912,A -85,B 0,C 180,E1 -10897.01,E2 -10897.01} C_VEL
LIN {X 0,Y 403.347,Z 837.548,A -85,B 0,C 180,E1 -10898.769,E2 -10898.769} C_VEL
LIN {X 0,Y 403.654,Z 830.605,A -85,B 0,C 180,E1 -10900.28,E2 -10900.28} C_VEL
LIN {X 0,Y 404.3,Z 821.968,A -85,B 0,C 180,E1 -10901.785,E2 -10901.785} C_VEL
LIN {X 0,Y 404.937,Z 813.074,A -85,B 0,C 180,E1 -10903.039,E2 -10903.039} C_VEL
LIN {X 0,Y 405.71,Z 801.178,A -85,B 0,C 180,E1 -10904.419,E2 -10904.419} C_VEL
LIN {X 0,Y 406.57,Z 790.488,A -85,B 0,C 180,E1 -10905.412,E2 -10905.412} C_VEL
LIN {X 0,Y 407.524,Z 778.494,A -85,B 0,C 180,E1 -10906.274,E2 -10906.274} C_VEL
LIN {X 0,Y 408.235,Z 765.999,A -85,B 0,C 180,E1 -10906.953,E2 -10906.953} C_VEL
LIN {X 0,Y 408.903,Z 753.823,A -85,B 0,C 180,E1 -10907.407,E2 -10907.407} C_VEL
LIN {X 0,Y 409.251,Z 738.475,A -85,B 0,C 180,E1 -10907.747,E2 -10907.747} C_VEL
LIN {X 0,Y 409.958,Z 669.706,A -85,B 0,C 180,E1 -10908.983,E2 -10908.983} C_VEL
LIN {X 0,Y 406.318,Z 638.711,A -85,B 0,C 180,E1 -10909.776,E2 -10909.776} C_VEL
LIN {X 0,Y 407.708,Z 616.996,A -85,B 0,C 180,E1 -10913.088,E2 -10913.088} C_VEL
LIN {X 0,Y 408.873,Z 601.632,A -85,B 0,C 180,E1 -10915.449,E2 -10915.449} C_VEL
LIN {X 0,Y 406.377,Z 589.309,A -85,B 0,C 180,E1 -10917.556,E2 -10917.556} C_VEL
LIN {X 0,Y 404.197,Z 580.138,A -85,B 0,C 180,E1 -10919.218,E2 -10919.218} C_VEL
LIN {X 0,Y 404.14,Z 580.143,A -85,B 0,C 180,E1 -10922.621,E2 -10922.621} C_VEL
LIN {X 0,Y 404.18,Z 580.136,A -85,B 0,C 180,E1 -10925.189,E2 -10925.189} C_VEL
LIN {X 0,Y 404.16,Z 580.137,A -85,B 0,C 180,E1 -10928.755,E2 -10928.755} C_VEL
LIN {X 0,Y 404.146,Z 580.14,A -85,B 0,C 180,E1 -10931.603,E2 -10931.603} C_VEL
LIN {X 0,Y 404.149,Z 580.139,A -85,B 0,C 180,E1 -10934.522,E2 -10934.522} C_VEL
LIN {X 0,Y 404.206,Z 580.132,A -85,B 0,C 180,E1 -10937.305,E2 -10937.305} C_VEL
LIN {X 0,Y 404.164,Z 580.135,A -85,B 0,C 180,E1 -10939.955,E2 -10939.955} C_VEL
LIN {X 0,Y 404.135,Z 580.141,A -85,B 0,C 180,E1 -10943.123,E2 -10943.123} C_VEL
LIN {X 0,Y 404.139,Z 580.135,A -85,B 0,C 180,E1 -10946.187,E2 -10946.187} C_VEL
LIN {X 0,Y 404.149,Z 580.138,A -85,B 0,C 180,E1 -10949.715,E2 -10949.715} C_VEL
LIN {X 0,Y 404.188,Z 580.134,A -85,B 0,C 180,E1 -10953.122,E2 -10953.122} C_VEL
LIN {X 0,Y 404.169,Z 580.135,A -85,B 0,C 180,E1 -10955.334,E2 -10955.334} C_VEL
LIN {X 0,Y 404.13,Z 580.138,A -85,B 0,C 180,E1 -10958.58,E2 -10958.58} C_VEL
LIN {X 0,Y 404.201,Z 580.132,A -85,B 0,C 180,E1 -10961.761,E2 -10961.761} C_VEL
LIN {X 0,Y 404.197,Z 580.128,A -85,B 0,C 180,E1 -10964.882,E2 -10964.882} C_VEL
LIN {X 0,Y 404.248,Z 580.128,A -85,B 0,C 180,E1 -10967.958,E2 -10967.958} C_VEL
LIN {X 0,Y 404.393,Z 580.098,A -85,B 0,C 180,E1 -10972.132,E2 -10972.132} C_VEL
LIN {X 0,Y 404.429,Z 580.104,A -85,B 0,C 180,E1 -10974.015,E2 -10974.015} C_VEL
LIN {X 0,Y 404.474,Z 580.089,A -85,B 0,C 180,E1 -10978.008,E2 -10978.008} C_VEL
LIN {X 0,Y 404.604,Z 580.076,A -85,B 0,C 180,E1 -10980,E2 -10980} C_VEL
LIN {X 0,Y 404.415,Z 580.107,A -85,B 0,C 180,E1 -10982.988,E2 -10982.988} C_VEL
LIN {X 0,Y 404.388,Z 580.1,A -85,B 0,C 180,E1 -10986.625,E2 -10986.625} C_VEL
LIN {X 0,Y 404.282,Z 580.128,A -85,B 0,C 180,E1 -10989.001,E2 -10989.001} C_VEL
LIN {X 0,Y 404.248,Z 580.118,A -85,B 0,C 180,E1 -10992.042,E2 -10992.042} C_VEL
LIN {X 0,Y 404.197,Z 580.138,A -85,B 0,C 180,E1 -10995.118,E2 -10995.118} C_VEL
LIN {X 0,Y 404.201,Z 580.127,A -85,B 0,C 180,E1 -10998.239,E2 -10998.239} C_VEL
LIN {X 0,Y 404.13,Z 580.144,A -85,B 0,C 180,E1 -11001.42,E2 -11001.42} C_VEL
LIN {X 0,Y 404.166,Z 580.131,A -85,B 0,C 180,E1 -11004.666,E2 -11004.666} C_VEL
LIN {X 0,Y 404.191,Z 580.134,A -85,B 0,C 180,E1 -11008,E2 -11008} C_VEL
LIN {X 0,Y 404.141,Z 580.143,A -85,B 0,C 180,E1 -11011.561,E2 -11011.561} C_VEL
LIN {X 0,Y 404.179,Z 580.133,A -85,B 0,C 180,E1 -11015.017,E2 -11015.017} C_VEL
LIN {X 0,Y 404.156,Z 580.141,A -85,B 0,C 180,E1 -11018.757,E2 -11018.757} C_VEL
LIN {X 0,Y 404.145,Z 580.121,A -85,B 0,C 180,E1 -11021.605,E2 -11021.605} C_VEL
LIN {X 0,Y 404.144,Z 580.14,A -85,B 0,C 180,E1 -11024.523,E2 -11024.523} C_VEL
LIN {X 0,Y 404.132,Z 580.132,A -85,B 0,C 180,E1 -11027.296,E2 -11027.296} C_VEL
LIN {X 0,Y 404.166,Z 580.14,A -85,B 0,C 180,E1 -11029.956,E2 -11029.956} C_VEL
LIN {X 0,Y 404.137,Z 580.14,A -85,B 0,C 180,E1 -11033.125,E2 -11033.125} C_VEL
LIN {X 0,Y 404.143,Z 580.142,A -85,B 0,C 180,E1 -11036.189,E2 -11036.189} C_VEL
LIN {X 0,Y 404.152,Z 580.142,A -85,B 0,C 180,E1 -11037.966,E2 -11037.966} C_VEL
LIN {X 0,Y 405.181,Z 583.064,A -85,B 0,C 180,E1 -11038.095,E2 -11038.095} C_VEL
LIN {X 0,Y 411.371,Z 597.46,A -85,B 0,C 180,E1 -11038.731,E2 -11038.731} C_VEL
LIN {X 0,Y 410.226,Z 681.356,A -85,B 0,C 180,E1 -11040.243,E2 -11040.243} C_VEL
LIN {X 0,Y 409.969,Z 693.787,A -85,B 0,C 180,E1 -11040.647,E2 -11040.647} C_VEL
LIN {X 0,Y 409.503,Z 706.71,A -85,B 0,C 180,E1 -11041.28,E2 -11041.28} C_VEL
LIN {X 0,Y 408.83,Z 718.56,A -85,B 0,C 180,E1 -11042.068,E2 -11042.068} C_VEL
LIN {X 0,Y 408.074,Z 729.325,A -85,B 0,C 180,E1 -11042.985,E2 -11042.985} C_VEL
LIN {X 0,Y 407.197,Z 739.667,A -85,B 0,C 180,E1 -11044.093,E2 -11044.093} C_VEL
LIN {X 0,Y 406.347,Z 749.952,A -85,B 0,C 180,E1 -11045.475,E2 -11045.475} C_VEL
LIN {X 0,Y 405.606,Z 758.029,A -85,B 0,C 180,E1 -11046.822,E2 -11046.822} C_VEL
LIN {X 0,Y 404.881,Z 765.417,A -85,B 0,C 180,E1 -11048.355,E2 -11048.355} C_VEL
LIN {X 0,Y 404.352,Z 771.058,A -85,B 0,C 180,E1 -11049.813,E2 -11049.813} C_VEL
LIN {X 0,Y 403.943,Z 775.414,A -85,B 0,C 180,E1 -11051.224,E2 -11051.224} C_VEL
LIN {X 0,Y 403.635,Z 779.098,A -85,B 0,C 180,E1 -11052.783,E2 -11052.783} C_VEL
LIN {X 0,Y 403.465,Z 780.972,A -85,B 0,C 180,E1 -11053.817,E2 -11053.817} C_VEL
LIN {X 0,Y 403.279,Z 782.371,A -85,B 0,C 180,E1 -11054.847,E2 -11054.847} C_VEL
LIN {X 0,Y 403.182,Z 783.337,A -85,B 0,C 180,E1 -11055.875,E2 -11055.875} C_VEL
LIN {X 0,Y 403.173,Z 784.021,A -85,B 0,C 180,E1 -11057.469,E2 -11057.469} C_VEL
LIN {X 0,Y 403.131,Z 783.777,A -85,B 0,C 180,E1 -11058.944,E2 -11058.944} C_VEL
LIN {X 0,Y 403.216,Z 782.063,A -85,B 0,C 180,E1 -11060.975,E2 -11060.975} C_VEL
LIN {X 0,Y 403.32,Z 780.553,A -85,B 0,C 180,E1 -11061.987,E2 -11061.987} C_VEL
LIN {X 0,Y 403.602,Z 777.875,A -85,B 0,C 180,E1 -11063.345,E2 -11063.345} C_VEL
LIN {X 0,Y 403.812,Z 773.427,A -85,B 0,C 180,E1 -11065.008,E2 -11065.008} C_VEL
LIN {X 0,Y 404.19,Z 767.224,A -85,B 0,C 180,E1 -11066.761,E2 -11066.761} C_VEL
LIN {X 0,Y 404.733,Z 760.42,A -85,B 0,C 180,E1 -11068.259,E2 -11068.259} C_VEL
LIN {X 0,Y 405.376,Z 751.923,A -85,B 0,C 180,E1 -11069.752,E2 -11069.752} C_VEL
LIN {X 0,Y 406.118,Z 742.795,A -85,B 0,C 180,E1 -11071.045,E2 -11071.045} C_VEL
LIN {X 0,Y 405.762,Z 738.43,A -85,B 0,C 180,E1 -11071.606,E2 -11071.606} C_VEL
LIN {X 0,Y 403.473,Z 731.109,A -85,B 0,C 180,E1 -11072.498,E2 -11072.498} C_VEL
LIN {X 0,Y 401.205,Z 723.401,A -85,B 0,C 180,E1 -11073.317,E2 -11073.317} C_VEL
LIN {X 0,Y 400.855,Z 718.327,A -85,B 0,C 180,E1 -11073.746,E2 -11073.746} C_VEL
LIN {X 0,Y 401.511,Z 705.681,A -85,B 0,C 180,E1 -11074.58,E2 -11074.58} C_VEL
LIN {X 0,Y 401.894,Z 693.29,A -85,B 0,C 180,E1 -11075.173,E2 -11075.173} C_VEL
LIN {X 0,Y 402.198,Z 680.489,A -85,B 0,C 180,E1 -11075.578,E2 -11075.578} C_VEL
LIN {X 0,Y 403.131,Z 597.307,A -85,B 0,C 180,E1 -11077.079,E2 -11077.079} C_VEL
LIN {X 0,Y 397.361,Z 581.052,A -85,B 0,C 180,E1 -11077.634,E2 -11077.634} C_VEL
LIN {X 0,Y 397.21,Z 581.004,A -85,B 0,C 180,E1 -11081.223,E2 -11081.223} C_VEL
LIN {X 0,Y 397.183,Z 581.011,A -85,B 0,C 180,E1 -11084.343,E2 -11084.343} C_VEL
LIN {X 0,Y 397.176,Z 581.01,A -85,B 0,C 180,E1 -11087.506,E2 -11087.506} C_VEL
LIN {X 0,Y 397.103,Z 581.016,A -85,B 0,C 180,E1 -11090.729,E2 -11090.729} C_VEL
LIN {X 0,Y 397.128,Z 581.02,A -85,B 0,C 180,E1 -11094.018,E2 -11094.018} C_VEL
LIN {X 0,Y 397.165,Z 581.013,A -85,B 0,C 180,E1 -11096.197,E2 -11096.197} C_VEL
LIN {X 0,Y 403.504,Z 598.048,A -85,B 0,C 180,E1 -11096.849,E2 -11096.849} C_VEL
LIN {X 0,Y 402.292,Z 682.117,A -85,B 0,C 180,E1 -11098.464,E2 -11098.464} C_VEL
LIN {X 0,Y 401.957,Z 695.976,A -85,B 0,C 180,E1 -11098.953,E2 -11098.953} C_VEL
LIN {X 0,Y 401.506,Z 707.792,A -85,B 0,C 180,E1 -11099.563,E2 -11099.563} C_VEL
LIN {X 0,Y 400.837,Z 720.036,A -85,B 0,C 180,E1 -11100.415,E2 -11100.415} C_VEL
LIN {X 0,Y 400.195,Z 730.786,A -85,B 0,C 180,E1 -11101.372,E2 -11101.372} C_VEL
LIN {X 0,Y 399.48,Z 740.773,A -85,B 0,C 180,E1 -11102.471,E2 -11102.471} C_VEL
LIN {X 0,Y 398.752,Z 750.005,A -85,B 0,C 180,E1 -11103.723,E2 -11103.723} C_VEL
LIN {X 0,Y 398.122,Z 757.753,A -85,B 0,C 180,E1 -11105.004,E2 -11105.004} C_VEL
LIN {X 0,Y 397.434,Z 765.763,A -85,B 0,C 180,E1 -11106.641,E2 -11106.641} C_VEL
LIN {X 0,Y 397.018,Z 772.101,A -85,B 0,C 180,E1 -11108.283,E2 -11108.283} C_VEL
LIN {X 0,Y 396.666,Z 776.198,A -85,B 0,C 180,E1 -11109.629,E2 -11109.629} C_VEL
LIN {X 0,Y 396.429,Z 779.462,A -85,B 0,C 180,E1 -11110.99,E2 -11110.99} C_VEL
LIN {X 0,Y 396.219,Z 781.98,A -85,B 0,C 180,E1 -11112.378,E2 -11112.378} C_VEL
LIN {X 0,Y 396.093,Z 783.746,A -85,B 0,C 180,E1 -11113.786,E2 -11113.786} C_VEL
LIN {X 0,Y 396.028,Z 784.724,A -85,B 0,C 180,E1 -11115.221,E2 -11115.221} C_VEL
LIN {X 0,Y 396.023,Z 784.893,A -85,B 0,C 180,E1 -11116.684,E2 -11116.684} C_VEL
LIN {X 0,Y 396.099,Z 784.229,A -85,B 0,C 180,E1 -11118.175,E2 -11118.175} C_VEL
LIN {X 0,Y 396.264,Z 782.665,A -85,B 0,C 180,E1 -11119.695,E2 -11119.695} C_VEL
LIN {X 0,Y 396.615,Z 779.245,A -85,B 0,C 180,E1 -11121.669,E2 -11121.669} C_VEL
LIN {X 0,Y 396.915,Z 775.988,A -85,B 0,C 180,E1 -11122.985,E2 -11122.985} C_VEL
LIN {X 0,Y 397.394,Z 770.41,A -85,B 0,C 180,E1 -11124.735,E2 -11124.735} C_VEL
LIN {X 0,Y 397.92,Z 764.82,A -85,B 0,C 180,E1 -11126.108,E2 -11126.108} C_VEL
LIN {X 0,Y 398.621,Z 757.178,A -85,B 0,C 180,E1 -11127.62,E2 -11127.62} C_VEL
LIN {X 0,Y 399.441,Z 748.349,A -85,B 0,C 180,E1 -11129.026,E2 -11129.026} C_VEL
LIN {X 0,Y 400.252,Z 738.795,A -85,B 0,C 180,E1 -11130.262,E2 -11130.262} C_VEL
LIN {X 0,Y 401.03,Z 728.047,A -85,B 0,C 180,E1 -11131.377,E2 -11131.377} C_VEL
LIN {X 0,Y 401.807,Z 715.908,A -85,B 0,C 180,E1 -11132.365,E2 -11132.365} C_VEL
LIN {X 0,Y 402.43,Z 704.661,A -85,B 0,C 180,E1 -11133.065,E2 -11133.065} C_VEL
LIN {X 0,Y 402.782,Z 691.892,A -85,B 0,C 180,E1 -11133.65,E2 -11133.65} C_VEL
LIN {X 0,Y 403.05,Z 679.487,A -85,B 0,C 180,E1 -11134.017,E2 -11134.017} C_VEL
LIN {X 0,Y 404.428,Z 598.83,A -85,B 0,C 180,E1 -11135.576,E2 -11135.576} C_VEL
LIN {X 0,Y 397.216,Z 581.565,A -85,B 0,C 180,E1 -11136.365,E2 -11136.365} C_VEL
LIN {X 0,Y 397.144,Z 581.016,A -85,B 0,C 180,E1 -11136.436,E2 -11136.436} C_VEL
LIN {X 0,Y 397.14,Z 581.019,A -85,B 0,C 180,E1 -11140.352,E2 -11140.352} C_VEL
LIN {X 0,Y 397.158,Z 581.012,A -85,B 0,C 180,E1 -11143.553,E2 -11143.553} C_VEL
LIN {X 0,Y 397.22,Z 581.007,A -85,B 0,C 180,E1 -11146.702,E2 -11146.702} C_VEL
LIN {X 0,Y 397.221,Z 581.005,A -85,B 0,C 180,E1 -11149.809,E2 -11149.809} C_VEL
LIN {X 0,Y 397.356,Z 580.989,A -85,B 0,C 180,E1 -11152.888,E2 -11152.888} C_VEL
LIN {X 0,Y 397.254,Z 581,A -85,B 0,C 180,E1 -11154.925,E2 -11154.925} C_VEL
LIN {X 0,Y 397.443,Z 580.974,A -85,B 0,C 180,E1 -11157.973,E2 -11157.973} C_VEL
LIN {X 0,Y 397.573,Z 580.961,A -85,B 0,C 180,E1 -11160,E2 -11160} C_VEL
LIN {X 0,Y 397.374,Z 580.981,A -85,B 0,C 180,E1 -11163.041,E2 -11163.041} C_VEL
LIN {X 0,Y 397.379,Z 580.985,A -85,B 0,C 180,E1 -11166.091,E2 -11166.091} C_VEL
LIN {X 0,Y 397.249,Z 580.996,A -85,B 0,C 180,E1 -11169.162,E2 -11169.162} C_VEL
LIN {X 0,Y 397.22,Z 581.003,A -85,B 0,C 180,E1 -11172.258,E2 -11172.258} C_VEL
LIN {X 0,Y 397.171,Z 581.005,A -85,B 0,C 180,E1 -11175.392,E2 -11175.392} C_VEL
LIN {X 0,Y 397.154,Z 581.013,A -85,B 0,C 180,E1 -11178.574,E2 -11178.574} C_VEL
LIN {X 0,Y 397.09,Z 581.017,A -85,B 0,C 180,E1 -11181.819,E2 -11181.819} C_VEL
LIN {X 0,Y 397.149,Z 581.013,A -85,B 0,C 180,E1 -11185.132,E2 -11185.132} C_VEL
LIN {X 0,Y 397.157,Z 581.007,A -85,B 0,C 180,E1 -11187.777,E2 -11187.777} C_VEL
LIN {X 0,Y 397.078,Z 581.021,A -85,B 0,C 180,E1 -11190.883,E2 -11190.883} C_VEL
LIN {X 0,Y 397.12,Z 581.018,A -85,B 0,C 180,E1 -11194.494,E2 -11194.494} C_VEL
LIN {X 0,Y 397.105,Z 581.022,A -85,B 0,C 180,E1 -11198.275,E2 -11198.275} C_VEL
LIN {X 0,Y 397.151,Z 581.011,A -85,B 0,C 180,E1 -11201.994,E2 -11201.994} C_VEL
LIN {X 0,Y 397.107,Z 581.02,A -85,B 0,C 180,E1 -11205.066,E2 -11205.066} C_VEL
LIN {X 0,Y 397.106,Z 581.02,A -85,B 0,C 180,E1 -11208.015,E2 -11208.015} C_VEL
LIN {X 0,Y 397.135,Z 581.017,A -85,B 0,C 180,E1 -11211.138,E2 -11211.138} C_VEL
LIN {X 0,Y 397.118,Z 581.02,A -85,B 0,C 180,E1 -11214.497,E2 -11214.497} C_VEL
LIN {X 0,Y 397.077,Z 581.027,A -85,B 0,C 180,E1 -11217.929,E2 -11217.929} C_VEL
LIN {X 0,Y 397.12,Z 581.14,A -85,B 0,C 180,E1 -11218.752,E2 -11218.752} C_VEL
LIN {X 0,Y 400,Z 593.677,A -85,B 0,C 180,E1 -11221.462,E2 -11221.462} C_VEL
LIN {X 0,Y 401.548,Z 602.227,A -85,B 0,C 180,E1 -11223.204,E2 -11223.204} C_VEL
LIN {X 0,Y 400.361,Z 616.852,A -85,B 0,C 180,E1 -11225.898,E2 -11225.898} C_VEL
LIN {X 0,Y 398.928,Z 637.563,A -85,B 0,C 180,E1 -11229.639,E2 -11229.639} C_VEL
LIN {X 0,Y 402.742,Z 665.7,A -85,B 0,C 180,E1 -11230.445,E2 -11230.445} C_VEL
LIN {X 0,Y 403.6,Z 675.079,A -85,B 0,C 180,E1 -11230.68,E2 -11230.68} C_VEL
LIN {X 0,Y 402.415,Z 748.495,A -85,B 0,C 180,E1 -11232.106,E2 -11232.106} C_VEL
LIN {X 0,Y 401.767,Z 762.12,A -85,B 0,C 180,E1 -11232.569,E2 -11232.569} C_VEL
LIN {X 0,Y 400.921,Z 774.544,A -85,B 0,C 180,E1 -11233.188,E2 -11233.188} C_VEL
LIN {X 0,Y 400.012,Z 787.332,A -85,B 0,C 180,E1 -11234.067,E2 -11234.067} C_VEL
LIN {X 0,Y 399.065,Z 798.748,A -85,B 0,C 180,E1 -11235.075,E2 -11235.075} C_VEL
LIN {X 0,Y 398.425,Z 808.43,A -85,B 0,C 180,E1 -11236.141,E2 -11236.141} C_VEL
LIN {X 0,Y 397.494,Z 818.42,A -85,B 0,C 180,E1 -11237.492,E2 -11237.492} C_VEL
LIN {X 0,Y 396.806,Z 827.559,A -85,B 0,C 180,E1 -11239.024,E2 -11239.024} C_VEL
LIN {X 0,Y 396.389,Z 834.937,A -85,B 0,C 180,E1 -11240.561,E2 -11240.561} C_VEL
LIN {X 0,Y 396.097,Z 841.681,A -85,B 0,C 180,E1 -11242.353,E2 -11242.353} C_VEL
LIN {X 0,Y 395.978,Z 846.164,A -85,B 0,C 180,E1 -11243.887,E2 -11243.887} C_VEL
LIN {X 0,Y 396.008,Z 848.559,A -85,B 0,C 180,E1 -11244.909,E2 -11244.909} C_VEL
LIN {X 0,Y 395.938,Z 850.474,A -85,B 0,C 180,E1 -11245.929,E2 -11245.929} C_VEL
LIN {X 0,Y 396.066,Z 851.94,A -85,B 0,C 180,E1 -11246.949,E2 -11246.949} C_VEL
LIN {X 0,Y 396.101,Z 852.988,A -85,B 0,C 180,E1 -11247.966,E2 -11247.966} C_VEL
LIN {X 0,Y 396.052,Z 853.626,A -85,B 0,C 180,E1 -11248.983,E2 -11248.983} C_VEL
LIN {X 0,Y 396.018,Z 853.827,A -85,B 0,C 180,E1 -11250,E2 -11250} C_VEL
LIN {X 0,Y 396.052,Z 853.606,A -85,B 0,C 180,E1 -11251.017,E2 -11251.017} C_VEL
LIN {X 0,Y 396.13,Z 852.987,A -85,B 0,C 180,E1 -11252.033,E2 -11252.033} C_VEL
LIN {X 0,Y 396.069,Z 851.952,A -85,B 0,C 180,E1 -11253.051,E2 -11253.051} C_VEL
LIN {X 0,Y 395.951,Z 850.449,A -85,B 0,C 180,E1 -11254.071,E2 -11254.071} C_VEL
LIN {X 0,Y 396,Z 847.389,A -85,B 0,C 180,E1 -11255.601,E2 -11255.601} C_VEL
LIN {X 0,Y 396.009,Z 843.228,A -85,B 0,C 180,E1 -11257.136,E2 -11257.136} C_VEL
LIN {X 0,Y 396.275,Z 836.841,A -85,B 0,C 180,E1 -11258.927,E2 -11258.927} C_VEL
LIN {X 0,Y 396.619,Z 829.877,A -85,B 0,C 180,E1 -11260.464,E2 -11260.464} C_VEL
LIN {X 0,Y 397.302,Z 821.203,A -85,B 0,C 180,E1 -11261.996,E2 -11261.996} C_VEL
LIN {X 0,Y 398.115,Z 810.865,A -85,B 0,C 180,E1 -11263.503,E2 -11263.503} C_VEL
LIN {X 0,Y 398.83,Z 800.986,A -85,B 0,C 180,E1 -11264.673,E2 -11264.673} C_VEL
LIN {X 0,Y 399.741,Z 790.411,A -85,B 0,C 180,E1 -11265.683,E2 -11265.683} C_VEL
LIN {X 0,Y 400.728,Z 778.6,A -85,B 0,C 180,E1 -11266.558,E2 -11266.558} C_VEL
LIN {X 0,Y 401.411,Z 767.613,A -85,B 0,C 180,E1 -11267.184,E2 -11267.184} C_VEL
LIN {X 0,Y 402.156,Z 754.63,A -85,B 0,C 180,E1 -11267.709,E2 -11267.709} C_VEL
LIN {X 0,Y 402.535,Z 742.204,A -85,B 0,C 180,E1 -11268.02,E2 -11268.02} C_VEL
LIN {X 0,Y 403.35,Z 670.374,A -85,B 0,C 180,E1 -11269.332,E2 -11269.332} C_VEL
LIN {X 0,Y 399.445,Z 637.543,A -85,B 0,C 180,E1 -11270.199,E2 -11270.199} C_VEL
LIN {X 0,Y 401.223,Z 612.442,A -85,B 0,C 180,E1 -11274.1,E2 -11274.1} C_VEL
LIN {X 0,Y 401.921,Z 602.624,A -85,B 0,C 180,E1 -11275.643,E2 -11275.643} C_VEL
LIN {X 0,Y 399.444,Z 590.584,A -85,B 0,C 180,E1 -11277.738,E2 -11277.738} C_VEL
LIN {X 0,Y 397.136,Z 581.018,A -85,B 0,C 180,E1 -11279.484,E2 -11279.484} C_VEL
LIN {X 0,Y 397.113,Z 581.018,A -85,B 0,C 180,E1 -11283.272,E2 -11283.272} C_VEL
